KUKA KRL program: MyProgram_252().src

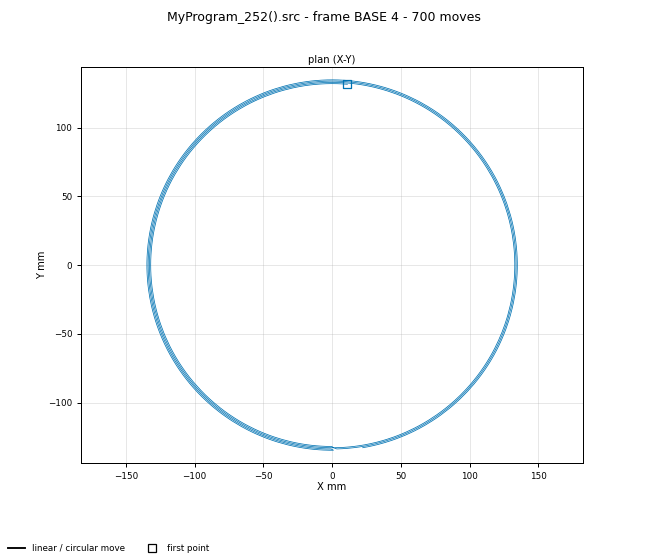
[picture p0: tool path of MyProgram_252().src in frame BASE 4, 700 of 700 moves have a stored position in this frame; points joined in program order, loops and branches not executed]
&ACCESS RVP
&REL 1
&PARAM TEMPLATE = C:\KRC\Roboter\Template\vorgabe
&PARAM EDITMASK = *
DEF MyProgram_252()
; ---- Setting reference (Base) ----
$BASE = BASE_DATA[4]

; --------------------------
; ---- Setting tool (TCP) ----
$TOOL = TOOL_DATA[3]
; --------------------------

$VEL.CP = VEL_APROX_PRINT
Startdeposition()
$VEL.CP = VEL_PRINT
LIN {X 11.0837,Y 131.5095,Z 165,A 85.1709,B 12.0272,C -0.0775,E1 12.0407,E2 365.1861} C_DIS
LIN {X 7.4461,Y 131.7673,Z 165,A 86.8868,B 12.0272,C -0.081,E1 12.0359,E2 363.4553} C_DIS
LIN {X 3.723,Y 131.9233,Z 165,A 88.4232,B 12.0272,C -0.079,E1 12.0316,E2 361.9291} C_DIS
LIN {X -0.4485,Y 131.9754,Z 165,A 90.2531,B 12.0272,C -0.0794,E1 12.0265,E2 360.0978} C_DIS
LIN {X -4.4864,Y 131.9012,Z 165,A 92.0505,B 12.0272,C -0.0802,E1 12.0215,E2 358.2962} C_DIS
LIN {X -8.3856,Y 131.7094,Z 165,A 93.7167,B 12.0272,C -0.0792,E1 12.0168,E2 356.6341} C_DIS
LIN {X -12.6017,Y 131.3727,Z 165,A 95.4316,B 12.0272,C -0.0756,E1 12.0121,E2 354.9346} C_DIS
LIN {X -16.1343,Y 130.9867,Z 165,A 97.1454,B 12.0272,C -0.0791,E1 12.0073,E2 353.2016} C_DIS
LIN {X -20.1878,Y 130.4225,Z 165,A 98.8102,B 12.0272,C -0.0756,E1 12.0027,E2 351.551} C_DIS
LIN {X -24.054,Y 129.7672,Z 165,A 100.47,B 12.0272,C -0.0736,E1 11.9982,E2 349.8973} C_DIS
LIN {X -28.8561,Y 128.7834,Z 165,A 102.7397,B 12.0272,C -0.0755,E1 11.992,E2 347.6125} C_DIS
LIN {X -32.281,Y 127.9668,Z 165,A 104.1599,B 12.0272,C -0.0718,E1 11.9881,E2 346.206} C_DIS
LIN {X -35.1769,Y 127.2017,Z 165,A 105.5524,B 12.0272,C -0.0729,E1 11.9844,E2 344.8037} C_DIS
LIN {X -39.2512,Y 126.0051,Z 165,A 107.686,B 12.0272,C -0.078,E1 11.9786,E2 342.6373} C_DIS
LIN {X -42.5812,Y 124.9193,Z 165,A 109.0037,B 12.0272,C -0.0717,E1 11.9752,E2 341.3448} C_DIS
LIN {X -46.1148,Y 123.6566,Z 165,A 110.4652,B 12.0272,C -0.066,E1 11.9714,E2 339.9042} C_DIS
LIN {X -48.8551,Y 122.6008,Z 165,A 111.8686,B 12.0272,C -0.0676,E1 11.9677,E2 338.4868} C_DIS
LIN {X -52.264,Y 121.1857,Z 165,A 113.1827,B 12.0273,C -0.0589,E1 11.9644,E2 337.2079} C_DIS
LIN {X -56.5408,Y 119.2509,Z 165,A 115.4801,B 12.0273,C -0.0623,E1 11.9585,E2 334.8819} C_DIS
LIN {X -59.5908,Y 117.7562,Z 165,A 116.8588,B 12.0273,C -0.0581,E1 11.9551,E2 333.5157} C_DIS
LIN {X -62.7217,Y 116.121,Z 165,A 118.4505,B 12.0273,C -0.0572,E1 11.9511,E2 331.9187} C_DIS
LIN {X -67.9902,Y 113.117,Z 165,A 121.2132,B 12.0273,C -0.0561,E1 11.9444,E2 329.1433} C_DIS
LIN {X -71.6438,Y 110.8388,Z 165,A 123.1109,B 12.0273,C -0.0537,E1 11.94,E2 327.2441} C_DIS
LIN {X -75.266,Y 108.4115,Z 165,A 124.9825,B 12.0273,C -0.05,E1 11.9357,E2 325.3769} C_DIS
LIN {X -78.4972,Y 106.096,Z 165,A 126.7552,B 12.0273,C -0.0479,E1 11.9316,E2 323.6005} C_DIS
LIN {X -81.8052,Y 103.5666,Z 165,A 128.5795,B 12.0273,C -0.0449,E1 11.9276,E2 321.7761} C_DIS
LIN {X -85.127,Y 100.8541,Z 165,A 130.4754,B 12.0274,C -0.0421,E1 11.9236,E2 319.878} C_DIS
LIN {X -88.4867,Y 97.9193,Z 165,A 132.4238,B 12.0274,C -0.0384,E1 11.9195,E2 317.9304} C_DIS
LIN {X -91.8671,Y 94.7546,Z 165,A 134.4232,B 12.0274,C -0.034,E1 11.9155,E2 315.9344} C_DIS
LIN {X -95.0357,Y 91.5768,Z 165,A 136.3955,B 12.0274,C -0.0303,E1 11.9116,E2 313.9614} C_DIS
LIN {X -98.0268,Y 88.3681,Z 165,A 138.3281,B 12.0274,C -0.0267,E1 11.908,E2 312.0276} C_DIS
LIN {X -100.8093,Y 85.18,Z 165,A 140.1811,B 12.0274,C -0.0229,E1 11.9046,E2 310.1748} C_DIS
LIN {X -103.4592,Y 81.9408,Z 165,A 142.0058,B 12.0274,C -0.0188,E1 11.9014,E2 308.3512} C_DIS
LIN {X -105.9833,Y 78.6485,Z 165,A 143.8053,B 12.0274,C -0.0144,E1 11.8984,E2 306.554} C_DIS
LIN {X -108.372,Y 75.3227,Z 165,A 145.6652,B 12.0274,C -0.0118,E1 11.8954,E2 304.6864} C_DIS
LIN {X -110.1166,Y 72.7488,Z 165,A 146.9884,B 12.0274,C -0.0079,E1 11.8933,E2 303.3679} C_DIS
LIN {X -114.2601,Y 66.0503,Z 165,A 150.4645,B 12.0274,C -0.0003,E1 11.8883,E2 299.8893} C_DIS
LIN {X -116.453,Y 62.1037,Z 165,A 152.4054,B 12.0274,C 0.0053,E1 11.8857,E2 297.953} C_DIS
LIN {X -118.178,Y 58.7502,Z 165,A 154.1788,B 12.0274,C 0.0066,E1 11.8835,E2 296.1653} C_DIS
LIN {X -120.2539,Y 54.3762,Z 165,A 155.9913,B 12.0274,C 0.0187,E1 11.8814,E2 294.3894} C_DIS
LIN {X -122.0747,Y 50.158,Z 165,A 158.225,B 12.0274,C 0.019,E1 11.8789,E2 292.1299} C_DIS
LIN {X -123.4373,Y 46.7004,Z 165,A 159.761,B 12.0274,C 0.0251,E1 11.8774,E2 290.605} C_DIS
LIN {X -124.6007,Y 43.5,Z 165,A 161.3273,B 12.0274,C 0.0274,E1 11.8759,E2 289.03} C_DIS
LIN {X -125.7157,Y 40.163,Z 165,A 162.8507,B 12.0274,C 0.0318,E1 11.8746,E2 287.5089} C_DIS
LIN {X -126.8783,Y 36.3323,Z 165,A 164.7046,B 12.0274,C 0.0343,E1 11.8731,E2 285.6434} C_DIS
LIN {X -127.9048,Y 32.5256,Z 165,A 166.3572,B 12.0274,C 0.0405,E1 11.872,E2 283.9996} C_DIS
LIN {X -129.1975,Y 26.9439,Z 165,A 168.886,B 12.0274,C 0.0468,E1 11.8704,E2 281.4689} C_DIS
LIN {X -129.8924,Y 23.3569,Z 165,A 170.4298,B 12.0274,C 0.0523,E1 11.8696,E2 279.9319} C_DIS
LIN {X -130.5188,Y 19.5658,Z 165,A 172.6918,B 12.0274,C 0.0443,E1 11.8687,E2 277.6013} C_DIS
LIN {X -131.1264,Y 14.9637,Z 165,A 174.1798,B 12.0274,C 0.0617,E1 11.8682,E2 276.1783} C_DIS
LIN {X -131.4859,Y 11.3639,Z 165,A 175.7627,B 12.0273,C 0.0661,E1 11.8678,E2 274.5957} C_DIS
LIN {X -131.7479,Y 7.761,Z 165,A 177.3281,B 12.0273,C 0.0708,E1 11.8675,E2 273.0324} C_DIS
LIN {X -131.9173,Y 3.9418,Z 165,A 178.9769,B 12.0273,C 0.0759,E1 11.8673,E2 271.3867} C_DIS
LIN {X -131.9786,Y 0.1809,Z 165,A -179.158,B 12.0273,C 0.0758,E1 11.8673,E2 269.4959} C_DIS
LIN {X -131.9226,Y -3.75,Z 165,A -177.5567,B 12.0272,C 0.0831,E1 11.8673,E2 267.9089} C_DIS
LIN {X -131.7465,Y -7.7839,Z 165,A -175.747,B 12.0272,C 0.087,E1 11.8676,E2 266.0943} C_DIS
LIN {X -131.4331,Y -11.9728,Z 165,A -173.8969,B 12.0272,C 0.0918,E1 11.8681,E2 264.243} C_DIS
LIN {X -130.9432,Y -16.4897,Z 165,A -171.415,B 12.0272,C 0.0864,E1 11.8689,E2 261.7023} C_DIS
LIN {X -130.292,Y -21.0255,Z 165,A -169.881,B 12.027,C 0.1022,E1 11.8696,E2 260.2248} C_DIS
LIN {X -129.8228,Y -23.746,Z 165,A -168.2147,B 12.0271,C 0.0954,E1 11.8705,E2 258.5036} C_DIS
LIN {X -128.9625,Y -28.0404,Z 165,A -166.7904,B 12.027,C 0.1113,E1 11.8712,E2 257.1383} C_DIS
LIN {X -127.9745,Y -32.2507,Z 165,A -164.9477,B 12.027,C 0.1174,E1 11.8724,E2 255.3015} C_DIS
LIN {X -127.1733,Y -35.2784,Z 165,A -163.2883,B 12.027,C 0.1147,E1 11.8737,E2 253.6076} C_DIS
LIN {X -125.8916,Y -39.6125,Z 165,A -161.4971,B 12.0268,C 0.1239,E1 11.8751,E2 251.8386} C_DIS
LIN {X -124.8136,Y -42.8859,Z 165,A -160.1385,B 12.0268,C 0.1311,E1 11.8763,E2 250.4977} C_DIS
LIN {X -123.7267,Y -45.9277,Z 165,A -158.7269,B 12.0268,C 0.1347,E1 11.8777,E2 249.0862} C_DIS
LIN {X -122.5757,Y -48.9172,Z 165,A -157.1757,B 12.0268,C 0.1349,E1 11.8793,E2 247.517} C_DIS
LIN {X -121.1996,Y -52.2318,Z 165,A -155.4885,B 12.0268,C 0.1362,E1 11.8811,E2 245.8156} C_DIS
LIN {X -118.0518,Y -59.0061,Z 165,A -152.363,B 12.0266,C 0.1474,E1 11.8849,E2 242.7068} C_DIS
LIN {X -116.1071,Y -62.7476,Z 165,A -150.4309,B 12.0266,C 0.1498,E1 11.8874,E2 240.764} C_DIS
LIN {X -113.9846,Y -66.5256,Z 165,A -148.5372,B 12.0266,C 0.1542,E1 11.89,E2 238.8701} C_DIS
LIN {X -111.9038,Y -69.9687,Z 165,A -146.721,B 12.0265,C 0.157,E1 11.8927,E2 237.0467} C_DIS
LIN {X -109.4503,Y -73.7476,Z 165,A -144.6081,B 12.0265,C 0.1581,E1 11.896,E2 234.9162} C_DIS
LIN {X -106.573,Y -77.8481,Z 165,A -142.5388,B 12.0264,C 0.1656,E1 11.8993,E2 232.8609} C_DIS
LIN {X -103.9034,Y -81.3764,Z 165,A -140.7404,B 12.0263,C 0.1727,E1 11.9024,E2 231.0783} C_DIS
LIN {X -101.0773,Y -84.861,Z 165,A -138.7731,B 12.0262,C 0.1766,E1 11.9059,E2 229.1097} C_DIS
LIN {X -95.5361,Y -91.0543,Z 165,A -135.0199,B 12.0262,C 0.1809,E1 11.913,E2 225.3409} C_DIS
LIN {X -92.3052,Y -94.328,Z 165,A -133.0328,B 12.0261,C 0.1851,E1 11.9169,E2 223.3559} C_DIS
LIN {X -89.3699,Y -97.1134,Z 165,A -131.2465,B 12.0261,C 0.1878,E1 11.9205,E2 221.5667} C_DIS
LIN {X -86.0304,Y -100.0839,Z 165,A -128.5328,B 12.0262,C 0.1733,E1 11.9265,E2 218.7596} C_DIS
LIN {X -81.3334,Y -103.9372,Z 165,A -126.6263,B 12.0259,C 0.195,E1 11.9305,E2 216.943} C_DIS
LIN {X -78.4155,Y -106.1561,Z 165,A -125.0015,B 12.0259,C 0.1969,E1 11.9341,E2 215.3146} C_DIS
LIN {X -75.3351,Y -108.3634,Z 165,A -123.2252,B 12.0259,C 0.1964,E1 11.9382,E2 213.5228} C_DIS
LIN {X -70.9431,Y -111.2886,Z 165,A -121.1913,B 12.0257,C 0.206,E1 11.9429,E2 211.5205} C_DIS
LIN {X -67.7985,Y -113.2318,Z 165,A -119.5058,B 12.0257,C 0.2063,E1 11.9469,E2 209.8255} C_DIS
LIN {X -64.4281,Y -115.1829,Z 165,A -117.8448,B 12.0257,C 0.2093,E1 11.9509,E2 208.1683} C_DIS
LIN {X -61.2678,Y -116.892,Z 165,A -116.2912,B 12.0257,C 0.2114,E1 11.9548,E2 206.6155} C_DIS
LIN {X -56.087,Y -119.4668,Z 165,A -113.7169,B 12.0257,C 0.2129,E1 11.9612,E2 204.0338} C_DIS
LIN {X -52.5475,Y -121.0631,Z 165,A -112.0714,B 12.0256,C 0.2157,E1 11.9654,E2 202.3931} C_DIS
LIN {X -49.413,Y -122.3759,Z 165,A -110.5286,B 12.0256,C 0.2155,E1 11.9694,E2 200.8422} C_DIS
LIN {X -45.5639,Y -123.863,Z 165,A -108.7403,B 12.0256,C 0.2173,E1 11.9741,E2 199.0541} C_DIS
LIN {X -41.8431,Y -125.1667,Z 165,A -107.0564,B 12.0256,C 0.2194,E1 11.9785,E2 197.3734} C_DIS
LIN {X -36.3101,Y -126.8847,Z 165,A -104.4227,B 12.0256,C 0.2183,E1 11.9856,E2 194.7251} C_DIS
LIN {X -30.1061,Y -128.4979,Z 165,A -101.6536,B 12.0255,C 0.2203,E1 11.9931,E2 191.9571} C_DIS
LIN {X -26.2294,Y -129.3429,Z 165,A -100.0343,B 12.0255,C 0.2237,E1 11.9975,E2 190.3499} C_DIS
LIN {X -22.4415,Y -130.0557,Z 165,A -98.2616,B 12.0255,C 0.2219,E1 12.0024,E2 188.5647} C_DIS
LIN {X -19.0063,Y -130.6004,Z 165,A -96.7818,B 12.0255,C 0.2231,E1 12.0065,E2 187.088} C_DIS
LIN {X -15.4939,Y -131.0631,Z 165,A -95.2317,B 12.0255,C 0.2231,E1 12.0108,E2 185.5359} C_DIS
LIN {X -11.5691,Y -131.4685,Z 165,A -93.6029,B 12.0254,C 0.2255,E1 12.0153,E2 183.9167} C_DIS
LIN {X -8.1546,Y -131.7236,Z 165,A -92.0385,B 12.0254,C 0.2236,E1 12.0197,E2 182.3422} C_DIS
LIN {X -4.1808,Y -131.9106,Z 165,A -90.2808,B 12.0254,C 0.2228,E1 12.0246,E2 180.5801} C_DIS
LIN {X -0.1658,Y -131.977,Z 165,A -88.5589,B 12.0254,C 0.2231,E1 12.0294,E2 178.86} C_DIS
LIN {X -0.1658,Y -131.977,Z 165,A -88.5589,B 12.0254,C 0.2231,E1 12.0294,E2 178.86} C_DIS
Enddeposition()
LIN {X 0.9669,Y -132.8884,Z 165,A -88.2437,B 12.0251,C 0.2348,E1 12.03,E2 178.6008} C_DIS
Startdeposition()
$VEL.CP = VEL_PRINT
LIN {X -1.6364,Y -132.8852,Z 165,A -89.9774,B 12.0248,C 0.2505,E1 12.025,E2 180.4097} C_DIS
LIN {X -5.3601,Y -132.7859,Z 165,A -91.5116,B 12.0248,C 0.2487,E1 12.0207,E2 181.9358} C_DIS
LIN {X -9.7113,Y -132.5386,Z 165,A -93.3724,B 12.0248,C 0.2482,E1 12.0156,E2 183.7952} C_DIS
LIN {X -13.4707,Y -132.2115,Z 165,A -95.1283,B 12.0248,C 0.2512,E1 12.0106,E2 185.5674} C_DIS
LIN {X -17.4667,Y -131.7411,Z 165,A -96.7577,B 12.0248,C 0.2482,E1 12.0061,E2 187.1846} C_DIS
LIN {X -21.5719,Y -131.1316,Z 165,A -98.5371,B 12.0248,C 0.2473,E1 12.0012,E2 188.9633} C_DIS
LIN {X -25.059,Y -130.5098,Z 165,A -100.049,B 12.0248,C 0.2464,E1 11.9971,E2 190.4738} C_DIS
LIN {X -28.736,Y -129.7516,Z 165,A -101.8197,B 12.0248,C 0.2493,E1 11.9922,E2 192.2633} C_DIS
LIN {X -33.8948,Y -128.499,Z 165,A -104.0819,B 12.0248,C 0.2473,E1 11.9861,E2 194.5228} C_DIS
LIN {X -37.8678,Y -127.3854,Z 165,A -105.8921,B 12.0248,C 0.2468,E1 11.9812,E2 196.337} C_DIS
LIN {X -41.8336,Y -126.1375,Z 165,A -107.5265,B 12.025,C 0.2416,E1 11.9769,E2 197.9525} C_DIS
LIN {X -45.0896,Y -125.0105,Z 165,A -109.037,B 12.025,C 0.2409,E1 11.9729,E2 199.4662} C_DIS
LIN {X -48.2888,Y -123.8099,Z 165,A -110.496,B 12.025,C 0.2392,E1 11.9691,E2 200.9235} C_DIS
LIN {X -51.3805,Y -122.5592,Z 165,A -111.9768,B 12.025,C 0.2388,E1 11.9653,E2 202.4095} C_DIS
LIN {X -54.4734,Y -121.2162,Z 165,A -113.4617,B 12.025,C 0.238,E1 11.9615,E2 203.8982} C_DIS
LIN {X -58.4379,Y -119.3559,Z 165,A -115.4331,B 12.025,C 0.2378,E1 11.9565,E2 205.8796} C_DIS
LIN {X -61.8393,Y -117.6289,Z 165,A -116.9935,B 12.0251,C 0.2337,E1 11.9527,E2 207.4296} C_DIS
LIN {X -65.5899,Y -115.5822,Z 165,A -118.9368,B 12.0251,C 0.2337,E1 11.9479,E2 209.385} C_DIS
LIN {X -70.5677,Y -112.6125,Z 165,A -121.3868,B 12.0252,C 0.229,E1 11.9421,E2 211.8288} C_DIS
LIN {X -74.0604,Y -110.3465,Z 165,A -123.3411,B 12.0252,C 0.23,E1 11.9374,E2 213.8019} C_DIS
LIN {X -77.5478,Y -107.9241,Z 165,A -125.115,B 12.0252,C 0.2258,E1 11.9334,E2 215.5685} C_DIS
LIN {X -80.4326,Y -105.7919,Z 165,A -126.629,B 12.0254,C 0.2224,E1 11.9301,E2 217.0782} C_DIS
LIN {X -83.8323,Y -103.1186,Z 165,A -128.8268,B 12.0253,C 0.2268,E1 11.9252,E2 219.3153} C_DIS
LIN {X -86.6745,Y -100.7408,Z 165,A -129.86,B 12.0256,C 0.2109,E1 11.9231,E2 220.2803} C_DIS
LIN {X -88.9595,Y -98.7297,Z 165,A -131.4614,B 12.0255,C 0.2151,E1 11.9197,E2 221.916} C_DIS
LIN {X -92.0207,Y -95.8825,Z 165,A -133.2607,B 12.0255,C 0.2116,E1 11.9161,E2 223.7142} C_DIS
LIN {X -95.158,Y -92.7701,Z 165,A -135.1993,B 12.0256,C 0.2085,E1 11.9122,E2 225.656} C_DIS
LIN {X -98.3035,Y -89.4294,Z 165,A -137.5582,B 12.0256,C 0.213,E1 11.9077,E2 228.0593} C_DIS
LIN {X -101.0067,Y -86.3653,Z 165,A -138.8103,B 12.0258,C 0.1977,E1 11.9055,E2 229.2498} C_DIS
LIN {X -103.1749,Y -83.7633,Z 165,A -140.4648,B 12.0258,C 0.1989,E1 11.9026,E2 230.9266} C_DIS
LIN {X -105.9003,Y -80.2895,Z 165,A -142.4027,B 12.0258,C 0.1953,E1 11.8992,E2 232.8676} C_DIS
LIN {X -108.5302,Y -76.6968,Z 165,A -144.5723,B 12.0258,C 0.1964,E1 11.8957,E2 235.0657} C_DIS
LIN {X -110.5325,Y -73.7818,Z 165,A -145.6225,B 12.026,C 0.1822,E1 11.8941,E2 236.0584} C_DIS
LIN {X -112.6635,Y -70.4857,Z 165,A -147.515,B 12.026,C 0.1826,E1 11.8912,E2 237.9739} C_DIS
LIN {X -114.7935,Y -66.9612,Z 165,A -149.3632,B 12.026,C 0.1798,E1 11.8886,E2 239.8295} C_DIS
LIN {X -116.8802,Y -63.2484,Z 165,A -151.2328,B 12.0261,C 0.1759,E1 11.8861,E2 241.7018} C_DIS
LIN {X -118.682,Y -59.7958,Z 165,A -152.8981,B 12.0261,C 0.1712,E1 11.884,E2 243.364} C_DIS
LIN {X -120.5344,Y -55.9658,Z 165,A -154.4185,B 12.0263,C 0.1595,E1 11.8822,E2 244.8456} C_DIS
LIN {X -121.5966,Y -53.6229,Z 165,A -155.7743,B 12.0263,C 0.162,E1 11.8806,E2 246.23} C_DIS
LIN {X -123.1001,Y -50.0721,Z 165,A -157.5682,B 12.0263,C 0.1604,E1 11.8786,E2 248.0382} C_DIS
LIN {X -124.4801,Y -46.5338,Z 165,A -159.1245,B 12.0264,C 0.1542,E1 11.8771,E2 249.5834} C_DIS
LIN {X -125.6277,Y -43.3406,Z 165,A -160.6042,B 12.0264,C 0.1505,E1 11.8757,E2 251.0639} C_DIS
LIN {X -126.7133,Y -40.0574,Z 165,A -162.2539,B 12.0264,C 0.1499,E1 11.8743,E2 252.7311} C_DIS
LIN {X -128.8623,Y -32.4851,Z 165,A -165.5463,B 12.0266,C 0.1381,E1 11.8719,E2 256.0083} C_DIS
LIN {X -129.7399,Y -28.7902,Z 165,A -167.6588,B 12.0266,C 0.1437,E1 11.8705,E2 258.1756} C_DIS
LIN {X -130.5159,Y -25.0267,Z 165,A -168.9735,B 12.0266,C 0.1315,E1 11.8699,E2 259.4482} C_DIS
LIN {X -131.4162,Y -19.7702,Z 165,A -171.4049,B 12.0267,C 0.1277,E1 11.8688,E2 261.893} C_DIS
LIN {X -132.0073,Y -15.3299,Z 165,A -173.2583,B 12.0267,C 0.1204,E1 11.8681,E2 263.7353} C_DIS
LIN {X -132.4193,Y -11.2216,Z 165,A -174.9858,B 12.0268,C 0.1141,E1 11.8677,E2 265.4546} C_DIS
LIN {X -132.6842,Y -7.4947,Z 165,A -176.7198,B 12.0268,C 0.112,E1 11.8674,E2 267.2015} C_DIS
LIN {X -132.8527,Y -3.3319,Z 165,A -178.5408,B 12.0269,C 0.1072,E1 11.8672,E2 269.0235} C_DIS
LIN {X -132.8939,Y 0.6025,Z 165,A 179.7573,B 12.0269,C 0.1023,E1 11.8672,E2 270.7243} C_DIS
LIN {X -132.7993,Y 5.017,Z 165,A 177.9002,B 12.027,C 0.0957,E1 11.8673,E2 272.5738} C_DIS
LIN {X -132.62,Y 8.5354,Z 165,A 176.3122,B 12.027,C 0.0927,E1 11.8676,E2 274.1682} C_DIS
LIN {X -132.3011,Y 12.5391,Z 165,A 174.6151,B 12.027,C 0.0868,E1 11.868,E2 275.8593} C_DIS
LIN {X -131.8994,Y 16.2346,Z 165,A 172.968,B 12.027,C 0.0831,E1 11.8685,E2 277.5099} C_DIS
LIN {X -130.8416,Y 23.2646,Z 165,A 169.7393,B 12.0271,C 0.0776,E1 11.87,E2 280.7543} C_DIS
LIN {X -129.8984,Y 28.0558,Z 165,A 167.27,B 12.0271,C 0.0793,E1 11.8714,E2 283.2638} C_DIS
LIN {X -128.9181,Y 32.2652,Z 165,A 166.0479,B 12.0272,C 0.0601,E1 11.8722,E2 284.4086} C_DIS
LIN {X -127.9808,Y 35.7998,Z 165,A 164.2862,B 12.0272,C 0.0596,E1 11.8734,E2 286.1902} C_DIS
LIN {X -127.0462,Y 38.9869,Z 165,A 162.8075,B 12.0272,C 0.0565,E1 11.8746,E2 287.6727} C_DIS
LIN {X -125.7951,Y 42.8579,Z 165,A 160.9368,B 12.0272,C 0.0541,E1 11.8763,E2 289.5552} C_DIS
LIN {X -124.4445,Y 46.629,Z 165,A 159.3402,B 12.0272,C 0.0464,E1 11.8778,E2 291.1344} C_DIS
LIN {X -123.1358,Y 49.9835,Z 165,A 157.7546,B 12.0273,C 0.0428,E1 11.8794,E2 292.7221} C_DIS
LIN {X -121.2066,Y 54.4949,Z 165,A 155.5761,B 12.0273,C 0.0384,E1 11.8819,E2 294.9055} C_DIS
LIN {X -118.7734,Y 59.6163,Z 165,A 153.1688,B 12.0273,C 0.031,E1 11.8848,E2 297.3056} C_DIS
LIN {X -116.5566,Y 63.8421,Z 165,A 150.5656,B 12.0273,C 0.0374,E1 11.8883,E2 299.9701} C_DIS
LIN {X -114.4892,Y 67.4793,Z 165,A 149.2931,B 12.0273,C 0.0212,E1 11.89,E2 301.1785} C_DIS
LIN {X -111.0541,Y 72.9943,Z 165,A 146.6881,B 12.0273,C 0.0098,E1 11.8939,E2 303.7573} C_DIS
LIN {X -108.206,Y 77.1537,Z 165,A 144.0936,B 12.0273,C 0.0137,E1 11.898,E2 306.3987} C_DIS
LIN {X -105.5046,Y 80.8083,Z 165,A 142.1364,B 12.0273,C 0.0089,E1 11.9013,E2 308.3535} C_DIS
LIN {X -102.8384,Y 84.1752,Z 165,A 140.2696,B 12.0273,C 0.0049,E1 11.9046,E2 310.22} C_DIS
LIN {X -99.9382,Y 87.5992,Z 165,A 138.3126,B 12.0273,C 0.001,E1 11.9081,E2 312.1774} C_DIS
LIN {X -96.9717,Y 90.8727,Z 165,A 136.3446,B 12.0273,C -0.0019,E1 11.9119,E2 314.1507} C_DIS
LIN {X -93.8909,Y 94.052,Z 165,A 134.4214,B 12.0273,C -0.0057,E1 11.9156,E2 316.0735} C_DIS
LIN {X -90.6399,Y 97.1885,Z 165,A 132.4789,B 12.0273,C -0.0098,E1 11.9196,E2 318.0133} C_DIS
LIN {X -87.2549,Y 100.2387,Z 165,A 130.5251,B 12.0273,C -0.014,E1 11.9236,E2 319.9637} C_DIS
LIN {X -83.8131,Y 103.1343,Z 165,A 128.5433,B 12.0273,C -0.0168,E1 11.9279,E2 321.9485} C_DIS
LIN {X -80.3503,Y 105.8544,Z 165,A 126.609,B 12.0273,C -0.0195,E1 11.9322,E2 323.885} C_DIS
LIN {X -76.857,Y 108.4172,Z 165,A 124.7384,B 12.0273,C -0.0228,E1 11.9364,E2 325.7541} C_DIS
LIN {X -73.2685,Y 110.8737,Z 165,A 122.8408,B 12.0273,C -0.0255,E1 11.9408,E2 327.6524} C_DIS
LIN {X -69.6079,Y 113.2076,Z 165,A 120.9734,B 12.0273,C -0.0286,E1 11.9452,E2 329.5175} C_DIS
LIN {X -65.7193,Y 115.5084,Z 165,A 118.2114,B 12.0273,C -0.0131,E1 11.9522,E2 332.3719} C_DIS
LIN {X -60.2277,Y 118.4622,Z 165,A 116.2852,B 12.0273,C -0.0343,E1 11.9567,E2 334.2074} C_DIS
LIN {X -52.6794,Y 122.0064,Z 165,A 112.8297,B 12.0273,C -0.0422,E1 11.9654,E2 337.6435} C_DIS
LIN {X -49.7383,Y 123.2346,Z 165,A 111.3701,B 12.0273,C -0.0418,E1 11.9692,E2 339.1121} C_DIS
LIN {X -46.1696,Y 124.6165,Z 165,A 109.7453,B 12.0273,C -0.0442,E1 11.9734,E2 340.7326} C_DIS
LIN {X -42.2829,Y 125.9879,Z 165,A 107.0728,B 12.0273,C -0.0252,E1 11.9808,E2 343.5074} C_DIS
LIN {X -36.2422,Y 127.8571,Z 165,A 105.3766,B 12.0273,C -0.0517,E1 11.985,E2 345.0822} C_DIS
LIN {X -32.1984,Y 128.935,Z 165,A 102.3456,B 12.0273,C -0.0243,E1 11.9936,E2 348.2541} C_DIS
LIN {X -25.1621,Y 130.4901,Z 165,A 100.5485,B 12.0273,C -0.0572,E1 11.9981,E2 349.8973} C_DIS
LIN {X -21.5719,Y 131.1316,Z 165,A 98.7353,B 12.0273,C -0.0524,E1 12.0032,E2 351.7378} C_DIS
LIN {X -18.2752,Y 131.6323,Z 165,A 97.1666,B 12.0273,C -0.0499,E1 12.0075,E2 353.3209} C_DIS
LIN {X -14.2264,Y 132.1302,Z 165,A 95.5011,B 12.0273,C -0.0529,E1 12.0121,E2 354.9744} C_DIS
LIN {X -10.2517,Y 132.4992,Z 165,A 93.7279,B 12.0273,C -0.0521,E1 12.0171,E2 356.7528} C_DIS
LIN {X -6.471,Y 132.7365,Z 165,A 92.1663,B 12.0273,C -0.0542,E1 12.0214,E2 358.3052} C_DIS
LIN {X -2.4477,Y 132.8717,Z 165,A 90.3952,B 12.0273,C -0.0536,E1 12.0264,E2 360.0796} C_DIS
LIN {X 1.5303,Y 132.8869,Z 165,A 88.6001,B 12.0273,C -0.0517,E1 12.0314,E2 361.8833} C_DIS
LIN {X 5.3663,Y 132.7857,Z 165,A 87.0553,B 12.0273,C -0.0544,E1 12.0357,E2 363.4145} C_DIS
LIN {X 9.3782,Y 132.5629,Z 165,A 85.2795,B 12.0273,C -0.0531,E1 12.0406,E2 365.1947} C_DIS
LIN {X 13.0895,Y 132.2482,Z 165,A 83.638,B 12.0273,C -0.0519,E1 12.0452,E2 366.8398} C_DIS
LIN {X 17.1232,Y 131.7861,Z 165,A 81.9542,B 12.0273,C -0.053,E1 12.0498,E2 368.5151} C_DIS
LIN {X 20.5913,Y 131.2891,Z 165,A 80.4758,B 12.0273,C -0.0532,E1 12.0539,E2 369.9893} C_DIS
LIN {X 24.4169,Y 130.6325,Z 165,A 78.7087,B 12.0273,C -0.0501,E1 12.0588,E2 371.767} C_DIS
LIN {X 28.2175,Y 129.8635,Z 165,A 76.8358,B 12.0273,C -0.0442,E1 12.064,E2 373.663} C_DIS
LIN {X 31.354,Y 129.1422,Z 165,A 75.6142,B 12.0273,C -0.0474,E1 12.0672,E2 374.8649} C_DIS
LIN {X 36.432,Y 127.804,Z 165,A 73.2336,B 12.0273,C -0.0429,E1 12.0737,E2 377.2588} C_DIS
LIN {X 40.5585,Y 126.5533,Z 165,A 71.654,B 12.0273,C -0.0484,E1 12.0778,E2 378.8054} C_DIS
LIN {X 43.6968,Y 125.5042,Z 165,A 70.2156,B 12.0273,C -0.0469,E1 12.0816,E2 380.245} C_DIS
LIN {X 46.7214,Y 124.4098,Z 165,A 68.8706,B 12.0273,C -0.0466,E1 12.0851,E2 381.585} C_DIS
LIN {X 49.9959,Y 123.1308,Z 165,A 67.3318,B 12.0273,C -0.0444,E1 12.0891,E2 383.1265} C_DIS
LIN {X 53.0238,Y 121.8575,Z 165,A 65.8769,B 12.0273,C -0.0419,E1 12.0929,E2 384.586} C_DIS
LIN {X 57.0972,Y 120.0025,Z 165,A 63.9663,B 12.0273,C -0.0401,E1 12.0977,E2 386.4943} C_DIS
LIN {X 60.7982,Y 118.1717,Z 165,A 62.2135,B 12.0273,C -0.0385,E1 12.1021,E2 388.2441} C_DIS
LIN {X 64.5473,Y 116.1674,Z 165,A 60.0014,B 12.0273,C -0.0262,E1 12.1076,E2 390.501} C_DIS
LIN {X 67.8292,Y 114.2823,Z 165,A 58.8108,B 12.0273,C -0.0353,E1 12.1104,E2 391.6399} C_DIS
LIN {X 71.1876,Y 112.2212,Z 165,A 56.9799,B 12.0273,C -0.0293,E1 12.1147,E2 393.4868} C_DIS
LIN {X 74.9013,Y 109.7776,Z 165,A 55.0661,B 12.0273,C -0.0263,E1 12.1192,E2 395.4006} C_DIS
LIN {X 78.4543,Y 107.2669,Z 165,A 53.2081,B 12.0273,C -0.0237,E1 12.1234,E2 397.257} C_DIS
LIN {X 82.0603,Y 104.5337,Z 165,A 51.2978,B 12.0273,C -0.0213,E1 12.1276,E2 399.1631} C_DIS
LIN {X 85.638,Y 101.6238,Z 165,A 49.3391,B 12.0273,C -0.0185,E1 12.1318,E2 401.1189} C_DIS
LIN {X 88.9555,Y 98.7332,Z 165,A 47.4128,B 12.0273,C -0.0141,E1 12.1358,E2 403.0494} C_DIS
LIN {X 92.1718,Y 95.7376,Z 165,A 45.5275,B 12.0273,C -0.0106,E1 12.1397,E2 404.9343} C_DIS
LIN {X 95.3263,Y 92.5965,Z 165,A 43.6368,B 12.0273,C -0.0074,E1 12.1434,E2 406.8225} C_DIS
LIN {X 98.4976,Y 89.2156,Z 165,A 41.6991,B 12.0273,C -0.0048,E1 12.147,E2 408.7538} C_DIS
LIN {X 101.4594,Y 85.8328,Z 165,A 39.7688,B 12.0273,C -0.0008,E1 12.1505,E2 410.6842} C_DIS
LIN {X 104.1879,Y 82.4995,Z 165,A 37.935,B 12.0273,C 0.0028,E1 12.1538,E2 412.5162} C_DIS
LIN {X 106.8542,Y 79.016,Z 165,A 36.0979,B 12.0273,C 0.0057,E1 12.1568,E2 414.348} C_DIS
LIN {X 109.8755,Y 74.7574,Z 165,A 34.1117,B 12.0273,C 0.0038,E1 12.16,E2 416.304} C_DIS
LIN {X 112.5366,Y 70.6879,Z 165,A 31.7528,B 12.0273,C 0.0161,E1 12.1636,E2 418.6956} C_DIS
LIN {X 116.3459,Y 64.2251,Z 165,A 28.7826,B 12.0273,C 0.017,E1 12.1677,E2 421.6366} C_DIS
LIN {X 117.7394,Y 61.6288,Z 165,A 26.8399,B 12.0273,C 0.0387,E1 12.1704,E2 423.6601} C_DIS
LIN {X 119.7761,Y 57.5713,Z 165,A 25.6457,B 12.0273,C 0.0229,E1 12.1717,E2 424.7651} C_DIS
LIN {X 121.5591,Y 53.7067,Z 165,A 23.621,B 12.0273,C 0.033,E1 12.1741,E2 426.8139} C_DIS
LIN {X 123.097,Y 50.0799,Z 165,A 21.7705,B 12.0273,C 0.0418,E1 12.1761,E2 428.6839} C_DIS
LIN {X 124.9887,Y 45.15,Z 165,A 19.6745,B 12.0273,C 0.043,E1 12.1781,E2 430.7603} C_DIS
LIN {X 126.1244,Y 41.8731,Z 165,A 17.6819,B 12.0273,C 0.0609,E1 12.18,E2 432.8134} C_DIS
LIN {X 127.481,Y 37.5413,Z 165,A 15.5908,B 12.0272,C 0.0702,E1 12.1816,E2 434.9222} C_DIS
LIN {X 128.8947,Y 32.3575,Z 165,A 14.0479,B 12.0272,C 0.0553,E1 12.1826,E2 436.3751} C_DIS
LIN {X 129.6644,Y 29.1222,Z 165,A 12.6402,B 12.0272,C 0.0586,E1 12.1835,E2 437.7811} C_DIS
LIN {X 130.2643,Y 26.3056,Z 165,A 11.3186,B 12.0272,C 0.0644,E1 12.1843,E2 439.1135} C_DIS
LIN {X 131.0478,Y 22.0743,Z 165,A 9.5249,B 12.0272,C 0.0681,E1 12.1851,E2 440.9016} C_DIS
LIN {X 131.5815,Y 18.631,Z 165,A 8.08,B 12.0272,C 0.0709,E1 12.1857,E2 442.3411} C_DIS
LIN {X 131.9753,Y 15.5986,Z 165,A 6.7469,B 12.0272,C 0.0751,E1 12.1862,E2 443.6773} C_DIS
LIN {X 132.3833,Y 11.6479,Z 165,A 4.9898,B 12.0272,C 0.0814,E1 12.1867,E2 445.4416} C_DIS
LIN {X 132.6429,Y 8.1647,Z 165,A 3.5534,B 12.0271,C 0.0839,E1 12.1869,E2 446.8712} C_DIS
LIN {X 132.804,Y 4.8961,Z 165,A 2.178,B 12.0271,C 0.0871,E1 12.1871,E2 448.2438} C_DIS
LIN {X 132.8903,Y 1.1306,Z 165,A 0.5737,B 12.0271,C 0.0913,E1 12.1871,E2 449.8476} C_DIS
LIN {X 132.8672,Y -2.7135,Z 165,A -1.1396,B 12.027,C 0.0978,E1 12.1871,E2 451.5694} C_DIS
LIN {X 132.7289,Y -6.6207,Z 165,A -2.7313,B 12.027,C 0.1001,E1 12.1869,E2 453.1516} C_DIS
LIN {X 132.4953,Y -10.305,Z 165,A -4.4267,B 12.027,C 0.1078,E1 12.1866,E2 454.8613} C_DIS
LIN {X 132.1415,Y -14.121,Z 165,A -5.945,B 12.0269,C 0.1089,E1 12.1862,E2 456.3652} C_DIS
LIN {X 131.7263,Y -17.5794,Z 165,A -7.4408,B 12.0269,C 0.1131,E1 12.1857,E2 457.8621} C_DIS
LIN {X 131.109,Y -21.7076,Z 165,A -9.218,B 12.0269,C 0.1178,E1 12.1849,E2 459.6387} C_DIS
LIN {X 130.5114,Y -25.0504,Z 165,A -10.6742,B 12.0268,C 0.1219,E1 12.1842,E2 461.0955} C_DIS
LIN {X 129.6726,Y -29.0862,Z 165,A -12.5338,B 12.0267,C 0.1294,E1 12.183,E2 462.9672} C_DIS
LIN {X 127.8249,Y -36.3574,Z 165,A -15.5263,B 12.0267,C 0.1319,E1 12.181,E2 465.9343} C_DIS
LIN {X 127.0711,Y -38.9055,Z 165,A -17.3413,B 12.0264,C 0.1539,E1 12.1794,E2 467.8312} C_DIS
LIN {X 125.5501,Y -43.5645,Z 165,A -18.4841,B 12.0267,C 0.1327,E1 12.1785,E2 468.8594} C_DIS
LIN {X 123.6469,Y -48.7082,Z 165,A -21.1249,B 12.0265,C 0.1472,E1 12.1759,E2 471.5366} C_DIS
LIN {X 122.5034,Y -51.514,Z 165,A -22.4443,B 12.0265,C 0.1512,E1 12.1745,E2 472.8591} C_DIS
LIN {X 121.1647,Y -54.5886,Z 165,A -24.148,B 12.0263,C 0.1624,E1 12.1725,E2 474.5958} C_DIS
LIN {X 118.2016,Y -60.7395,Z 165,A -26.7453,B 12.0263,C 0.1607,E1 12.1693,E2 477.1546} C_DIS
LIN {X 116.7166,Y -63.5486,Z 165,A -28.3209,B 12.0262,C 0.1701,E1 12.1672,E2 478.7568} C_DIS
LIN {X 114.5191,Y -67.4284,Z 165,A -29.9563,B 12.0262,C 0.1671,E1 12.165,E2 480.3598} C_DIS
LIN {X 112.637,Y -70.5282,Z 165,A -31.6494,B 12.0262,C 0.1748,E1 12.1625,E2 482.0704} C_DIS
LIN {X 110.4141,Y -73.9591,Z 165,A -33.3857,B 12.0261,C 0.1785,E1 12.1598,E2 483.8056} C_DIS
LIN {X 108.0253,Y -77.4063,Z 165,A -35.1776,B 12.0261,C 0.1825,E1 12.1569,E2 485.5976} C_DIS
LIN {X 105.5493,Y -80.7497,Z 165,A -36.983,B 12.0259,C 0.1872,E1 12.1539,E2 487.4065} C_DIS
LIN {X 102.7009,Y -84.3434,Z 165,A -39.2897,B 12.0257,C 0.201,E1 12.1498,E2 489.7554} C_DIS
LIN {X 100.14,Y -87.368,Z 165,A -40.5908,B 12.0258,C 0.1938,E1 12.1475,E2 491.0091} C_DIS
LIN {X 97.3535,Y -90.4627,Z 165,A -42.4198,B 12.0258,C 0.1988,E1 12.144,E2 492.8442} C_DIS
LIN {X 93.2409,Y -94.6963,Z 165,A -45.0926,B 12.0256,C 0.2079,E1 12.1387,E2 495.5354} C_DIS
LIN {X 89.4924,Y -98.2464,Z 165,A -47.1594,B 12.0256,C 0.2082,E1 12.1345,E2 497.5853} C_DIS
LIN {X 86.2368,Y -101.116,Z 165,A -49.3072,B 12.0254,C 0.2195,E1 12.1299,E2 499.7685} C_DIS
LIN {X 83.3123,Y -103.5387,Z 165,A -50.7256,B 12.0254,C 0.2168,E1 12.1269,E2 501.1622} C_DIS
LIN {X 79.7827,Y -106.2827,Z 165,A -52.5102,B 12.0254,C 0.2166,E1 12.123,E2 502.9316} C_DIS
LIN {X 76.2834,Y -108.8218,Z 165,A -54.3684,B 12.0254,C 0.2198,E1 12.1187,E2 504.7909} C_DIS
LIN {X 70.5979,Y -112.5934,Z 165,A -57.332,B 12.0253,C 0.2255,E1 12.1118,E2 507.7601} C_DIS
LIN {X 66.8243,Y -114.8729,Z 165,A -59.164,B 12.0253,C 0.2267,E1 12.1074,E2 509.5856} C_DIS
LIN {X 63.1793,Y -116.9174,Z 165,A -60.9618,B 12.0253,C 0.2294,E1 12.103,E2 511.3847} C_DIS
LIN {X 60.1113,Y -118.5214,Z 165,A -62.374,B 12.0253,C 0.2294,E1 12.0995,E2 512.7883} C_DIS
LIN {X 56.7026,Y -120.1911,Z 165,A -63.9919,B 12.0252,C 0.2313,E1 12.0955,E2 514.4056} C_DIS
LIN {X 53.9423,Y -121.4538,Z 165,A -65.2668,B 12.0252,C 0.2321,E1 12.0922,E2 515.6775} C_DIS
LIN {X 50.9073,Y -122.7568,Z 165,A -66.6995,B 12.0252,C 0.2341,E1 12.0885,E2 517.1125} C_DIS
LIN {X 47.8283,Y -123.9889,Z 165,A -68.1466,B 12.0251,C 0.2363,E1 12.0848,E2 518.5628} C_DIS
LIN {X 44.4901,Y -125.2266,Z 165,A -70.3388,B 12.0247,C 0.2553,E1 12.0788,E2 520.8358} C_DIS
LIN {X 39.5333,Y -126.8789,Z 165,A -71.8407,B 12.0251,C 0.238,E1 12.075,E2 522.2488} C_DIS
LIN {X 36.3429,Y -127.8289,Z 165,A -73.8534,B 12.0247,C 0.2544,E1 12.0694,E2 524.3325} C_DIS
LIN {X 32.0909,Y -128.9623,Z 165,A -75.3708,B 12.0249,C 0.2462,E1 12.0654,E2 525.8054} C_DIS
LIN {X 27.4918,Y -130.0196,Z 165,A -77.3499,B 12.0249,C 0.2463,E1 12.0601,E2 527.7793} C_DIS
LIN {X 23.4369,Y -130.8108,Z 165,A -79.0304,B 12.0249,C 0.2449,E1 12.0555,E2 529.4486} C_DIS
LIN {X 19.9627,Y -131.3864,Z 165,A -80.625,B 12.0249,C 0.2478,E1 12.051,E2 531.0535} C_DIS
LIN {X 15.8832,Y -131.9413,Z 165,A -82.3086,B 12.0249,C 0.2464,E1 12.0464,E2 532.7271} C_DIS
LIN {X 12.5231,Y -132.3026,Z 165,A -83.8155,B 12.0249,C 0.2483,E1 12.0422,E2 534.2409} C_DIS
LIN {X 8.3124,Y -132.6338,Z 165,A -85.6164,B 12.0249,C 0.2484,E1 12.0372,E2 536.0404} C_DIS
LIN {X 4.4295,Y -132.822,Z 165,A -87.3781,B 12.0249,C 0.251,E1 12.0322,E2 537.8134} C_DIS
LIN {X 0.9669,Y -132.8884,Z 165,A -88.2416,B 12.0251,C 0.2353,E1 12.0301,E2 538.6008} C_DIS
Enddeposition()
LIN {X 0.9669,Y -132.8884,Z 165,A -88.2416,B 12.0251,C 0.2353,E1 12.0301,E2 538.6008} C_DIS
Startdeposition()
$VEL.CP = VEL_PRINT
LIN {X 3.4476,Y -133.7679,Z 165,A -86.8697,B 11.7259,C 0.2508,E1 11.7348,E2 537.3149} C_DIS
LIN {X 7.4151,Y -133.6083,Z 165,A -85.1128,B 11.7259,C 0.2489,E1 11.7397,E2 535.5501} C_DIS
LIN {X 11.5039,Y -133.3168,Z 165,A -83.4137,B 11.7259,C 0.2497,E1 11.7444,E2 533.8569} C_DIS
LIN {X 15.6993,Y -132.8879,Z 165,A -81.6455,B 11.7259,C 0.2498,E1 11.7493,E2 532.0923} C_DIS
LIN {X 19.6622,Y -132.3615,Z 165,A -79.8699,B 11.7259,C 0.2473,E1 11.7542,E2 530.3078} C_DIS
LIN {X 23.6313,Y -131.7087,Z 165,A -78.2236,B 11.7259,C 0.2481,E1 11.7587,E2 528.6697} C_DIS
LIN {X 27.7651,Y -130.9005,Z 165,A -76.4185,B 11.7259,C 0.2468,E1 11.7637,E2 526.8632} C_DIS
LIN {X 31.1356,Y -130.1392,Z 165,A -74.9659,B 11.7259,C 0.2463,E1 11.7676,E2 525.4129} C_DIS
LIN {X 37.917,Y -128.3276,Z 165,A -72.297,B 11.7259,C 0.2524,E1 11.7747,E2 522.7836} C_DIS
LIN {X 44.9586,Y -126.0337,Z 165,A -68.7539,B 11.7261,C 0.2393,E1 11.7842,E2 519.192} C_DIS
LIN {X 48.2636,Y -124.8048,Z 165,A -67.2556,B 11.7261,C 0.2379,E1 11.7881,E2 517.6939} C_DIS
LIN {X 52.0084,Y -123.2919,Z 165,A -65.4551,B 11.7262,C 0.2338,E1 11.7928,E2 515.8832} C_DIS
LIN {X 55.8704,Y -121.59,Z 165,A -63.8487,B 11.7262,C 0.2367,E1 11.7968,E2 514.3001} C_DIS
LIN {X 59.1064,Y -120.0499,Z 165,A -62.3529,B 11.7262,C 0.2356,E1 11.8006,E2 512.8077} C_DIS
LIN {X 61.8554,Y -118.6574,Z 165,A -60.943,B 11.7262,C 0.2313,E1 11.8041,E2 511.3854} C_DIS
LIN {X 65.6882,Y -116.5811,Z 165,A -59.0186,B 11.7264,C 0.2269,E1 11.8088,E2 509.4521} C_DIS
LIN {X 69.4893,Y -114.3564,Z 165,A -57.1431,B 11.7264,C 0.2241,E1 11.8133,E2 507.5761} C_DIS
LIN {X 72.5091,Y -112.4648,Z 165,A -55.2494,B 11.7266,C 0.2115,E1 11.8179,E2 505.635} C_DIS
LIN {X 76.0644,Y -110.0928,Z 165,A -53.7756,B 11.7266,C 0.2179,E1 11.8212,E2 504.2038} C_DIS
LIN {X 79.6574,Y -107.5214,Z 165,A -51.8327,B 11.7266,C 0.2131,E1 11.8256,E2 502.2527} C_DIS
LIN {X 83.2485,Y -104.7653,Z 165,A -49.4161,B 11.7269,C 0.1962,E1 11.831,E2 499.7743} C_DIS
LIN {X 87.3744,Y -101.3497,Z 165,A -47.7425,B 11.7267,C 0.2086,E1 11.8344,E2 498.1757} C_DIS
LIN {X 92.1853,Y -96.9952,Z 165,A -45.1397,B 11.7267,C 0.2076,E1 11.8397,E2 495.5918} C_DIS
LIN {X 96.8673,Y -92.3191,Z 165,A -42.1943,B 11.7269,C 0.1984,E1 11.8456,E2 492.6295} C_DIS
LIN {X 98.8979,Y -90.1407,Z 165,A -40.7322,B 11.7269,C 0.1904,E1 11.8484,E2 491.1427} C_DIS
LIN {X 103.1778,Y -85.2082,Z 165,A -38.1449,B 11.727,C 0.1896,E1 11.853,E2 488.5783} C_DIS
LIN {X 106.0329,Y -81.6288,Z 165,A -36.1689,B 11.727,C 0.1845,E1 11.8564,E2 486.5982} C_DIS
LIN {X 108.7062,Y -78.0325,Z 165,A -34.2904,B 11.7271,C 0.1809,E1 11.8595,E2 484.7224} C_DIS
LIN {X 111.2021,Y -74.4324,Z 165,A -32.4529,B 11.7271,C 0.1772,E1 11.8624,E2 482.8875} C_DIS
LIN {X 113.5966,Y -70.7239,Z 165,A -30.6217,B 11.7272,C 0.174,E1 11.8651,E2 481.0614} C_DIS
LIN {X 116.4701,Y -65.8857,Z 165,A -28.165,B 11.7274,C 0.1664,E1 11.8686,E2 478.5962} C_DIS
LIN {X 118.5447,Y -62.0701,Z 165,A -26.468,B 11.7274,C 0.166,E1 11.8708,E2 476.917} C_DIS
LIN {X 120.2214,Y -58.7586,Z 165,A -24.3731,B 11.7276,C 0.1476,E1 11.8734,E2 474.7575} C_DIS
LIN {X 122.0802,Y -54.7903,Z 165,A -23.0646,B 11.7275,C 0.1584,E1 11.8749,E2 473.5172} C_DIS
LIN {X 123.3727,Y -51.815,Z 165,A -21.6187,B 11.7275,C 0.1529,E1 11.8765,E2 472.0628} C_DIS
LIN {X 124.8321,Y -48.1934,Z 165,A -19.8872,B 11.7276,C 0.1466,E1 11.8782,E2 470.3219} C_DIS
LIN {X 126.2272,Y -44.4143,Z 165,A -17.8082,B 11.7278,C 0.1318,E1 11.8802,E2 468.197} C_DIS
LIN {X 127.5834,Y -40.3507,Z 165,A -16.3675,B 11.7278,C 0.1377,E1 11.8814,E2 466.803} C_DIS
LIN {X 129.9789,Y -31.8006,Z 165,A -12.6537,B 11.7278,C 0.1292,E1 11.8841,E2 463.0959} C_DIS
LIN {X 130.8308,Y -28.0877,Z 165,A -11.0824,B 11.7278,C 0.1262,E1 11.885,E2 461.5301} C_DIS
LIN {X 131.6622,Y -23.8911,Z 165,A -9.3284,B 11.7278,C 0.123,E1 11.886,E2 459.7836} C_DIS
LIN {X 132.2177,Y -20.5943,Z 165,A -7.9094,B 11.7279,C 0.1191,E1 11.8866,E2 458.3645} C_DIS
LIN {X 132.7345,Y -16.9524,Z 165,A -6.2245,B 11.7279,C 0.1114,E1 11.8872,E2 456.6644} C_DIS
LIN {X 133.1755,Y -13.0379,Z 165,A -4.6438,B 11.728,C 0.1094,E1 11.8877,E2 455.0949} C_DIS
LIN {X 133.5131,Y -8.971,Z 165,A -2.8297,B 11.728,C 0.1024,E1 11.8881,E2 453.2707} C_DIS
LIN {X 133.7145,Y -5.1103,Z 165,A -1.3034,B 11.728,C 0.1011,E1 11.8882,E2 451.7583} C_DIS
LIN {X 133.8093,Y -1.0017,Z 165,A 0.4017,B 11.7281,C 0.0975,E1 11.8883,E2 450.0581} C_DIS
LIN {X 133.7823,Y 2.9034,Z 165,A 2.162,B 11.7281,C 0.0901,E1 11.8883,E2 448.2852} C_DIS
LIN {X 133.6607,Y 6.3724,Z 165,A 3.5705,B 11.7281,C 0.0879,E1 11.8881,E2 446.8846} C_DIS
LIN {X 133.4217,Y 10.2248,Z 165,A 5.2743,B 11.7282,C 0.0816,E1 11.8877,E2 445.1729} C_DIS
LIN {X 133.0741,Y 14.0364,Z 165,A 6.8213,B 11.7282,C 0.0793,E1 11.8873,E2 443.6355} C_DIS
LIN {X 132.5974,Y 17.9983,Z 165,A 8.5088,B 11.7282,C 0.075,E1 11.8867,E2 441.9489} C_DIS
LIN {X 132.0059,Y 21.9109,Z 165,A 10.1326,B 11.7283,C 0.072,E1 11.886,E2 440.3321} C_DIS
LIN {X 131.4343,Y 25.1122,Z 165,A 11.5362,B 11.7283,C 0.0677,E1 11.8853,E2 438.9258} C_DIS
LIN {X 130.6191,Y 29.0656,Z 165,A 13.3786,B 11.7283,C 0.0595,E1 11.8842,E2 437.0678} C_DIS
LIN {X 129.5964,Y 33.3249,Z 165,A 15.4061,B 11.7284,C 0.05,E1 11.8828,E2 435.0199} C_DIS
LIN {X 128.6655,Y 36.7605,Z 165,A 17.0729,B 11.7284,C 0.0417,E1 11.8815,E2 433.3342} C_DIS
LIN {X 127.4545,Y 40.7544,Z 165,A 18.481,B 11.7284,C 0.0473,E1 11.8804,E2 431.971} C_DIS
LIN {X 126.0065,Y 45.034,Z 165,A 20.0785,B 11.7284,C 0.0513,E1 11.8789,E2 430.4131} C_DIS
LIN {X 125.1236,Y 47.4332,Z 165,A 21.4833,B 11.7284,C 0.0397,E1 11.8775,E2 428.9696} C_DIS
LIN {X 123.4807,Y 51.5563,Z 165,A 23.1062,B 11.7284,C 0.0422,E1 11.8759,E2 427.3789} C_DIS
LIN {X 122.2386,Y 54.4363,Z 165,A 24.5762,B 11.7284,C 0.0351,E1 11.8742,E2 425.8924} C_DIS
LIN {X 120.7723,Y 57.6159,Z 165,A 26.6563,B 11.7285,C 0.0151,E1 11.8716,E2 423.7399} C_DIS
LIN {X 118.5198,Y 62.1175,Z 165,A 28.0575,B 11.7285,C 0.0304,E1 11.8699,E2 422.4295} C_DIS
LIN {X 114.9933,Y 68.4296,Z 165,A 31.289,B 11.7285,C 0.0189,E1 11.8655,E2 419.1796} C_DIS
LIN {X 112.7858,Y 72.0101,Z 165,A 33.0905,B 11.7285,C 0.0144,E1 11.8628,E2 417.3769} C_DIS
LIN {X 110.7764,Y 75.0643,Z 165,A 34.5286,B 11.7285,C 0.0141,E1 11.8606,E2 415.9533} C_DIS
LIN {X 108.119,Y 78.8447,Z 165,A 36.6247,B 11.7285,C 0.0063,E1 11.8571,E2 413.8418} C_DIS
LIN {X 105.4547,Y 82.3741,Z 165,A 38.491,B 11.7285,C 0.0027,E1 11.854,E2 411.9777} C_DIS
LIN {X 102.7164,Y 85.7642,Z 165,A 40.3641,B 11.7285,C -0.0017,E1 11.8506,E2 410.1028} C_DIS
LIN {X 99.6877,Y 89.266,Z 165,A 42.2779,B 11.7285,C -0.0042,E1 11.8471,E2 408.1963} C_DIS
LIN {X 96.5849,Y 92.6146,Z 165,A 44.2369,B 11.7285,C -0.0084,E1 11.8434,E2 406.2359} C_DIS
LIN {X 93.4271,Y 95.7996,Z 165,A 46.1537,B 11.7285,C -0.0122,E1 11.8396,E2 404.3188} C_DIS
LIN {X 90.2223,Y 98.8239,Z 165,A 48.0358,B 11.7285,C -0.0157,E1 11.8357,E2 402.4366} C_DIS
LIN {X 86.9129,Y 101.7462,Z 165,A 49.9029,B 11.7285,C -0.0187,E1 11.8318,E2 400.5716} C_DIS
LIN {X 83.4779,Y 104.5827,Z 165,A 51.7846,B 11.7285,C -0.0214,E1 11.8277,E2 398.6924} C_DIS
LIN {X 79.8844,Y 107.3524,Z 165,A 53.6956,B 11.7285,C -0.024,E1 11.8234,E2 396.7847} C_DIS
LIN {X 76.1746,Y 110.0163,Z 165,A 55.5504,B 11.7285,C -0.0245,E1 11.8192,E2 394.9417} C_DIS
LIN {X 72.5881,Y 112.415,Z 165,A 57.4903,B 11.7285,C -0.0298,E1 11.8147,E2 392.9903} C_DIS
LIN {X 68.8184,Y 114.7616,Z 165,A 59.4521,B 11.7285,C -0.0342,E1 11.81,E2 391.0208} C_DIS
LIN {X 64.0121,Y 117.5097,Z 165,A 61.6997,B 11.7285,C -0.0343,E1 11.8045,E2 388.7879} C_DIS
LIN {X 60.0573,Y 119.5791,Z 165,A 63.6898,B 11.7285,C -0.0388,E1 11.7996,E2 386.7881} C_DIS
LIN {X 55.5824,Y 121.7232,Z 165,A 65.701,B 11.7285,C -0.0384,E1 11.7945,E2 384.7905} C_DIS
LIN {X 51.883,Y 123.3443,Z 165,A 67.4214,B 11.7285,C -0.0401,E1 11.7901,E2 383.0711} C_DIS
LIN {X 48.4835,Y 124.7193,Z 165,A 68.8848,B 11.7285,C -0.039,E1 11.7863,E2 381.6207} C_DIS
LIN {X 45.3998,Y 125.8746,Z 165,A 70.2857,B 11.7285,C -0.0402,E1 11.7827,E2 380.2209} C_DIS
LIN {X 42.3412,Y 126.9362,Z 165,A 71.6332,B 11.7285,C -0.0404,E1 11.7791,E2 378.8782} C_DIS
LIN {X 38.4289,Y 128.1771,Z 165,A 73.5808,B 11.7285,C -0.0466,E1 11.7739,E2 376.9081} C_DIS
LIN {X 34.6432,Y 129.2496,Z 165,A 75.1784,B 11.7285,C -0.0457,E1 11.7696,E2 375.3212} C_DIS
LIN {X 28.9241,Y 130.6503,Z 165,A 77.7866,B 11.7285,C -0.0494,E1 11.7625,E2 372.7031} C_DIS
LIN {X 25.031,Y 131.4499,Z 165,A 79.3614,B 11.7285,C -0.0471,E1 11.7582,E2 371.144} C_DIS
LIN {X 21.0482,Y 132.1474,Z 165,A 81.0678,B 11.7285,C -0.0472,E1 11.7535,E2 369.4411} C_DIS
LIN {X 17.4584,Y 132.6682,Z 165,A 82.5986,B 11.7285,C -0.0472,E1 11.7493,E2 367.9134} C_DIS
LIN {X 13.9741,Y 133.0808,Z 165,A 84.2034,B 11.7285,C -0.0502,E1 11.7448,E2 366.2968} C_DIS
LIN {X 9.9199,Y 133.4439,Z 165,A 85.831,B 11.7285,C -0.0477,E1 11.7403,E2 364.6837} C_DIS
LIN {X 6.5787,Y 133.6503,Z 165,A 87.338,B 11.7285,C -0.0496,E1 11.7361,E2 363.1684} C_DIS
LIN {X 2.3208,Y 133.792,Z 165,A 89.1626,B 11.7285,C -0.0496,E1 11.731,E2 361.3446} C_DIS
LIN {X -1.9465,Y 133.7982,Z 165,A 91.01,B 11.7285,C -0.05,E1 11.7258,E2 359.4957} C_DIS
LIN {X -6.0463,Y 133.6771,Z 165,A 92.8219,B 11.7285,C -0.0511,E1 11.7208,E2 357.678} C_DIS
LIN {X -9.8448,Y 133.4494,Z 165,A 94.3701,B 11.7285,C -0.0487,E1 11.7165,E2 356.1404} C_DIS
LIN {X -14.053,Y 133.0723,Z 165,A 96.1471,B 11.7285,C -0.0473,E1 11.7116,E2 354.3682} C_DIS
LIN {X -17.325,Y 132.6856,Z 165,A 97.6078,B 11.7285,C -0.0479,E1 11.7075,E2 352.9024} C_DIS
LIN {X -21.1327,Y 132.1343,Z 165,A 99.2948,B 11.7285,C -0.048,E1 11.7028,E2 351.2118} C_DIS
LIN {X -25.3626,Y 131.3865,Z 165,A 102.2629,B 11.7283,C -0.0739,E1 11.6944,E2 348.1085} C_DIS
LIN {X -33.1086,Y 129.6512,Z 165,A 104.4277,B 11.7284,C -0.0419,E1 11.6889,E2 346.0952} C_DIS
LIN {X -35.5537,Y 129.003,Z 165,A 106.5323,B 11.7284,C -0.0652,E1 11.6829,E2 343.8684} C_DIS
LIN {X -41.9852,Y 127.0547,Z 165,A 108.5659,B 11.7284,C -0.0425,E1 11.6778,E2 341.9389} C_DIS
LIN {X -46.3447,Y 125.5313,Z 165,A 110.5391,B 11.7284,C -0.0403,E1 11.6726,E2 339.9679} C_DIS
LIN {X -49.9539,Y 124.1376,Z 165,A 112.0908,B 11.7284,C -0.036,E1 11.6686,E2 338.4299} C_DIS
LIN {X -56.1455,Y 121.4628,Z 165,A 114.9775,B 11.7284,C -0.0324,E1 11.6612,E2 335.546} C_DIS
LIN {X -59.0223,Y 120.0913,Z 165,A 116.2782,B 11.7284,C -0.0291,E1 11.6579,E2 334.2541} C_DIS
LIN {X -65.994,Y 116.4087,Z 165,A 119.9127,B 11.7284,C -0.03,E1 11.649,E2 330.5921} C_DIS
LIN {X -69.9504,Y 114.0745,Z 165,A 121.854,B 11.7284,C -0.0264,E1 11.6443,E2 328.6557} C_DIS
LIN {X -73.7871,Y 111.6314,Z 165,A 123.7771,B 11.7284,C -0.0226,E1 11.6398,E2 326.7374} C_DIS
LIN {X -77.4046,Y 109.1545,Z 165,A 125.6942,B 11.7285,C -0.0202,E1 11.6354,E2 324.8175} C_DIS
LIN {X -80.8869,Y 106.5996,Z 165,A 127.5839,B 11.7285,C -0.0178,E1 11.6312,E2 322.9248} C_DIS
LIN {X -84.3715,Y 103.8637,Z 165,A 129.5256,B 11.7285,C -0.0152,E1 11.6269,E2 320.9796} C_DIS
LIN {X -87.7343,Y 101.0389,Z 165,A 131.4036,B 11.7285,C -0.0114,E1 11.623,E2 319.1039} C_DIS
LIN {X -91.012,Y 98.0966,Z 165,A 133.3039,B 11.7285,C -0.0079,E1 11.619,E2 317.2039} C_DIS
LIN {X -94.2167,Y 95.0226,Z 165,A 135.2147,B 11.7285,C -0.0041,E1 11.6152,E2 315.294} C_DIS
LIN {X -97.3982,Y 91.7587,Z 165,A 137.1509,B 11.7285,C 0.0005,E1 11.6115,E2 313.3618} C_DIS
LIN {X -100.3945,Y 88.4706,Z 165,A 139.0811,B 11.7285,C 0.0042,E1 11.6079,E2 311.4306} C_DIS
LIN {X -103.2492,Y 85.1219,Z 165,A 140.9885,B 11.7285,C 0.008,E1 11.6045,E2 309.5226} C_DIS
LIN {X -106.0153,Y 81.6516,Z 165,A 142.9621,B 11.7285,C 0.0109,E1 11.6011,E2 307.5423} C_DIS
LIN {X -108.6932,Y 78.0507,Z 165,A 144.8621,B 11.7285,C 0.016,E1 11.5979,E2 305.6471} C_DIS
LIN {X -111.1696,Y 74.481,Z 165,A 146.5952,B 11.7285,C 0.0234,E1 11.5952,E2 303.9313} C_DIS
LIN {X -114.3797,Y 69.4506,Z 165,A 149.1988,B 11.7285,C 0.0289,E1 11.5914,E2 301.3249} C_DIS
LIN {X -116.1133,Y 66.5119,Z 165,A 151.0539,B 11.7285,C 0.0241,E1 11.5887,E2 299.4242} C_DIS
LIN {X -117.7902,Y 63.4946,Z 165,A 152.388,B 11.7285,C 0.0311,E1 11.587,E2 298.1092} C_DIS
LIN {X -120.0244,Y 59.158,Z 165,A 154.2962,B 11.7285,C 0.0405,E1 11.5846,E2 296.2249} C_DIS
LIN {X -121.7452,Y 55.5348,Z 165,A 156.3971,B 11.7285,C 0.0369,E1 11.5821,E2 294.0801} C_DIS
LIN {X -123.1566,Y 52.3323,Z 165,A 157.7164,B 11.7285,C 0.0449,E1 11.5806,E2 292.7841} C_DIS
LIN {X -124.6428,Y 48.6802,Z 165,A 159.3045,B 11.7285,C 0.0517,E1 11.579,E2 291.21} C_DIS
LIN {X -125.7463,Y 45.7557,Z 165,A 160.6648,B 11.7284,C 0.055,E1 11.5777,E2 289.8485} C_DIS
LIN {X -126.8939,Y 42.4681,Z 165,A 162.1244,B 11.7284,C 0.0599,E1 11.5764,E2 288.3944} C_DIS
LIN {X -127.858,Y 39.4717,Z 165,A 163.4924,B 11.7284,C 0.0633,E1 11.5752,E2 287.0256} C_DIS
LIN {X -128.7597,Y 36.4237,Z 165,A 164.9443,B 11.7284,C 0.0652,E1 11.5741,E2 285.5644} C_DIS
LIN {X -129.888,Y 32.1758,Z 165,A 166.9032,B 11.7284,C 0.069,E1 11.5727,E2 283.5984} C_DIS
LIN {X -130.7464,Y 28.4785,Z 165,A 168.4712,B 11.7283,C 0.0749,E1 11.5718,E2 282.039} C_DIS
LIN {X -131.5678,Y 24.4143,Z 165,A 171.1287,B 11.7283,C 0.061,E1 11.5704,E2 279.2768} C_DIS
LIN {X -132.5657,Y 18.2331,Z 165,A 173.0366,B 11.7283,C 0.0856,E1 11.5697,E2 277.4658} C_DIS
LIN {X -133.022,Y 14.5202,Z 165,A 174.5988,B 11.7282,C 0.0912,E1 11.5692,E2 275.9101} C_DIS
LIN {X -133.3597,Y 10.9961,Z 165,A 176.1736,B 11.7282,C 0.0944,E1 11.5688,E2 274.3299} C_DIS
LIN {X -133.6268,Y 7.0471,Z 165,A 177.8602,B 11.7282,C 0.0995,E1 11.5685,E2 272.646} C_DIS
LIN {X -133.7686,Y 3.4224,Z 165,A 179.5307,B 11.7281,C 0.1016,E1 11.5683,E2 270.963} C_DIS
LIN {X -133.8116,Y -0.6599,Z 165,A -178.7517,B 11.7281,C 0.1074,E1 11.5683,E2 269.2511} C_DIS
LIN {X -133.7212,Y -4.9389,Z 165,A -176.9514,B 11.728,C 0.1135,E1 11.5685,E2 267.4566} C_DIS
LIN {X -133.5503,Y -8.3667,Z 165,A -175.4608,B 11.728,C 0.1174,E1 11.5687,E2 265.965} C_DIS
LIN {X -133.2319,Y -12.4511,Z 165,A -173.6538,B 11.728,C 0.1214,E1 11.5691,E2 264.1534} C_DIS
LIN {X -132.8363,Y -16.1322,Z 165,A -172.044,B 11.7279,C 0.1255,E1 11.5697,E2 262.5422} C_DIS
LIN {X -132.0586,Y -21.5946,Z 165,A -169.6887,B 11.7278,C 0.1325,E1 11.5706,E2 260.1901} C_DIS
LIN {X -130.6754,Y -28.8077,Z 165,A -166.5325,B 11.7277,C 0.1413,E1 11.5724,E2 257.0357} C_DIS
LIN {X -129.9663,Y -31.8529,Z 165,A -164.2801,B 11.7279,C 0.1252,E1 11.574,E2 254.6731} C_DIS
LIN {X -128.353,Y -37.8305,Z 165,A -162.4367,B 11.7276,C 0.1503,E1 11.5753,E2 252.9308} C_DIS
LIN {X -127.0751,Y -41.924,Z 165,A -160.5616,B 11.7276,C 0.1545,E1 11.5769,E2 251.0527} C_DIS
LIN {X -126.0161,Y -45.0074,Z 165,A -159.1728,B 11.7275,C 0.1585,E1 11.5782,E2 249.6659} C_DIS
LIN {X -124.8859,Y -48.0549,Z 165,A -157.7851,B 11.7275,C 0.1624,E1 11.5795,E2 248.2798} C_DIS
LIN {X -123.5832,Y -51.3109,Z 165,A -156.2489,B 11.7274,C 0.1657,E1 11.5812,E2 246.7407} C_DIS
LIN {X -121.8783,Y -55.2419,Z 165,A -154.2389,B 11.7274,C 0.1667,E1 11.5835,E2 244.7108} C_DIS
LIN {X -119.4296,Y -60.351,Z 165,A -151.9989,B 11.7272,C 0.1771,E1 11.5862,E2 242.4952} C_DIS
LIN {X -117.6766,Y -63.706,Z 165,A -150.182,B 11.7272,C 0.1769,E1 11.5886,E2 240.6557} C_DIS
LIN {X -115.4351,Y -67.6818,Z 165,A -148.2564,B 11.7272,C 0.1824,E1 11.5913,E2 238.7349} C_DIS
LIN {X -113.4231,Y -71.0028,Z 165,A -146.4972,B 11.7271,C 0.1844,E1 11.5939,E2 236.965} C_DIS
LIN {X -111.0266,Y -74.6947,Z 165,A -144.4867,B 11.7271,C 0.1861,E1 11.597,E2 234.9403} C_DIS
LIN {X -107.9772,Y -79.0382,Z 165,A -142.3465,B 11.7269,C 0.1943,E1 11.6005,E2 232.8177} C_DIS
LIN {X -105.2904,Y -82.5833,Z 165,A -140.4795,B 11.7269,C 0.1995,E1 11.6036,E2 230.9563} C_DIS
LIN {X -102.764,Y -85.7074,Z 165,A -138.6694,B 11.7269,C 0.2012,E1 11.6069,E2 229.1361} C_DIS
LIN {X -98.1093,Y -90.9982,Z 165,A -135.6323,B 11.7267,C 0.2072,E1 11.6125,E2 226.0981} C_DIS
LIN {X -94.9324,Y -94.3074,Z 165,A -133.6806,B 11.7267,C 0.2114,E1 11.6163,E2 224.1487} C_DIS
LIN {X -91.6891,Y -97.4639,Z 165,A -131.7393,B 11.7266,C 0.2151,E1 11.6202,E2 222.2078} C_DIS
LIN {X -88.4452,Y -100.4169,Z 165,A -129.8281,B 11.7266,C 0.2179,E1 11.6242,E2 220.2933} C_DIS
LIN {X -86.1176,Y -102.4199,Z 165,A -128.1718,B 11.7266,C 0.2124,E1 11.6279,E2 218.5954} C_DIS
LIN {X -83.052,Y -104.9216,Z 165,A -126.7773,B 11.7264,C 0.2223,E1 11.6308,E2 217.2383} C_DIS
LIN {X -80.3516,Y -107.0036,Z 165,A -125.3282,B 11.7264,C 0.225,E1 11.634,E2 215.791} C_DIS
LIN {X -77.4756,Y -109.1044,Z 165,A -123.6453,B 11.7264,C 0.2238,E1 11.6379,E2 214.089} C_DIS
LIN {X -73.2597,Y -111.9787,Z 165,A -121.5913,B 11.7263,C 0.2302,E1 11.6426,E2 212.0515} C_DIS
LIN {X -69.9067,Y -114.1013,Z 165,A -119.7126,B 11.7263,C 0.2284,E1 11.6472,E2 210.151} C_DIS
LIN {X -65.3769,Y -116.756,Z 165,A -117.7752,B 11.7261,C 0.2388,E1 11.6518,E2 208.2521} C_DIS
LIN {X -62.411,Y -118.3657,Z 165,A -116.2544,B 11.7261,C 0.2388,E1 11.6555,E2 206.7221} C_DIS
LIN {X -58.6004,Y -120.2995,Z 165,A -114.354,B 11.7261,C 0.2394,E1 11.6603,E2 204.8131} C_DIS
LIN {X -54.8888,Y -122.0362,Z 165,A -112.626,B 11.7261,C 0.242,E1 11.6647,E2 203.0883} C_DIS
LIN {X -51.7465,Y -123.4013,Z 165,A -111.1627,B 11.7261,C 0.2436,E1 11.6684,E2 201.6255} C_DIS
LIN {X -48.3364,Y -124.7765,Z 165,A -109.6406,B 11.726,C 0.2463,E1 11.6724,E2 200.1098} C_DIS
LIN {X -45.2262,Y -125.9372,Z 165,A -108.2504,B 11.726,C 0.2483,E1 11.676,E2 198.7233} C_DIS
LIN {X -41.4632,Y -127.2281,Z 165,A -106.3498,B 11.726,C 0.245,E1 11.6811,E2 196.7982} C_DIS
LIN {X -37.8361,Y -128.3513,Z 165,A -104.7933,B 11.726,C 0.2478,E1 11.6852,E2 195.2499} C_DIS
LIN {X -32.0791,Y -129.9118,Z 165,A -102.1285,B 11.726,C 0.2467,E1 11.6925,E2 192.5711} C_DIS
LIN {X -28.0756,Y -130.8334,Z 165,A -100.4658,B 11.7259,C 0.25,E1 11.697,E2 190.9199} C_DIS
LIN {X -23.8847,Y -131.6633,Z 165,A -98.6277,B 11.7259,C 0.2505,E1 11.702,E2 189.0802} C_DIS
LIN {X -19.9916,Y -132.311,Z 165,A -96.8762,B 11.7259,C 0.2496,E1 11.7069,E2 187.3205} C_DIS
LIN {X -16.1672,Y -132.8321,Z 165,A -95.2849,B 11.7259,C 0.2515,E1 11.7113,E2 185.7362} C_DIS
LIN {X -12.448,Y -133.2322,Z 165,A -93.6675,B 11.7259,C 0.2513,E1 11.7158,E2 184.1163} C_DIS
LIN {X -8.3899,Y -133.5489,Z 165,A -91.9623,B 11.7259,C 0.2524,E1 11.7205,E2 182.4151} C_DIS
LIN {X -4.4631,Y -133.7397,Z 165,A -90.1944,B 11.7259,C 0.2503,E1 11.7255,E2 180.636} C_DIS
LIN {X -0.6045,Y -133.8108,Z 165,A -88.6563,B 11.7259,C 0.253,E1 11.7297,E2 179.1113} C_DIS
LIN {X -0.6045,Y -133.8108,Z 165,A -88.6563,B 11.7259,C 0.253,E1 11.7297,E2 179.1113} C_DIS
Enddeposition()
LIN {X 0.9754,Y -134.7225,Z 165,A -88.2276,B 11.6439,C 0.2704,E1 11.6492,E2 178.7721} C_DIS
Startdeposition()
$VEL.CP = VEL_PRINT
LIN {X -2.16,Y -134.7129,Z 165,A -89.9303,B 11.6437,C 0.2798,E1 11.6443,E2 180.5213} C_DIS
LIN {X -6.4439,Y -134.5764,Z 165,A -91.7954,B 11.6437,C 0.2809,E1 11.639,E2 182.3924} C_DIS
LIN {X -10.1253,Y -134.3495,Z 165,A -93.3383,B 11.6437,C 0.2802,E1 11.6348,E2 183.9328} C_DIS
LIN {X -13.8716,Y -134.0152,Z 165,A -94.9459,B 11.6437,C 0.2802,E1 11.6303,E2 185.542} C_DIS
LIN {X -17.4813,Y -133.5911,Z 165,A -96.4307,B 11.6437,C 0.2783,E1 11.6262,E2 187.0198} C_DIS
LIN {X -20.6896,Y -133.132,Z 165,A -97.8664,B 11.6437,C 0.2793,E1 11.6222,E2 188.463} C_DIS
LIN {X -24.9374,Y -132.4025,Z 165,A -99.7057,B 11.6437,C 0.2787,E1 11.6171,E2 190.3037} C_DIS
LIN {X -28.4662,Y -131.6884,Z 165,A -101.2055,B 11.6437,C 0.2772,E1 11.6131,E2 191.8} C_DIS
LIN {X -32.3626,Y -130.7878,Z 165,A -103.1219,B 11.6437,C 0.2815,E1 11.6078,E2 193.7432} C_DIS
LIN {X -36.652,Y -129.6492,Z 165,A -104.7088,B 11.6438,C 0.273,E1 11.6036,E2 195.2935} C_DIS
LIN {X -39.2733,Y -128.8788,Z 165,A -106.0143,B 11.6438,C 0.2756,E1 11.6001,E2 196.6169} C_DIS
LIN {X -42.7819,Y -127.7571,Z 165,A -107.5215,B 11.6438,C 0.273,E1 11.5961,E2 198.117} C_DIS
LIN {X -46.0717,Y -126.6083,Z 165,A -108.981,B 11.6438,C 0.2712,E1 11.5922,E2 199.5739} C_DIS
LIN {X -49.1604,Y -125.4412,Z 165,A -110.4533,B 11.6438,C 0.2715,E1 11.5884,E2 201.0547} C_DIS
LIN {X -52.7712,Y -123.9672,Z 165,A -112.0523,B 11.644,C 0.2684,E1 11.5843,E2 202.6465} C_DIS
LIN {X -55.2591,Y -122.8763,Z 165,A -113.245,B 11.644,C 0.268,E1 11.5812,E2 203.8437} C_DIS
LIN {X -58.4551,Y -121.3889,Z 165,A -114.8516,B 11.644,C 0.2688,E1 11.5771,E2 205.4634} C_DIS
LIN {X -62.0951,Y -119.5686,Z 165,A -116.5756,B 11.644,C 0.2666,E1 11.5728,E2 207.1865} C_DIS
LIN {X -65.9349,Y -117.4956,Z 165,A -118.4478,B 11.644,C 0.2645,E1 11.5683,E2 209.0606} C_DIS
LIN {X -72.3718,Y -113.6444,Z 165,A -121.4073,B 11.6443,C 0.2547,E1 11.5613,E2 211.9915} C_DIS
LIN {X -74.8218,Y -112.046,Z 165,A -122.9273,B 11.6442,C 0.2591,E1 11.5576,E2 213.545} C_DIS
LIN {X -78.4947,Y -109.5044,Z 165,A -124.7882,B 11.6442,C 0.2552,E1 11.5534,E2 215.4009} C_DIS
LIN {X -81.8218,Y -107.0411,Z 165,A -126.6053,B 11.6442,C 0.2536,E1 11.5493,E2 217.2244} C_DIS
LIN {X -85.5704,Y -104.0696,Z 165,A -128.4839,B 11.6444,C 0.2465,E1 11.5453,E2 219.0834} C_DIS
LIN {X -87.905,Y -102.1044,Z 165,A -129.9705,B 11.6444,C 0.2484,E1 11.5421,E2 220.5926} C_DIS
LIN {X -91.3174,Y -99.0645,Z 165,A -131.9113,B 11.6444,C 0.2447,E1 11.5381,E2 222.5324} C_DIS
LIN {X -94.582,Y -95.953,Z 165,A -133.8662,B 11.6445,C 0.2418,E1 11.5341,E2 224.491} C_DIS
LIN {X -97.7218,Y -92.7536,Z 165,A -135.8258,B 11.6445,C 0.2391,E1 11.5303,E2 226.4562} C_DIS
LIN {X -100.8681,Y -89.3211,Z 165,A -137.7074,B 11.6447,C 0.2327,E1 11.5268,E2 228.3249} C_DIS
LIN {X -103.3934,Y -86.3858,Z 165,A -139.4092,B 11.6447,C 0.2303,E1 11.5237,E2 230.0326} C_DIS
LIN {X -105.9905,Y -83.1784,Z 165,A -141.1692,B 11.6448,C 0.2265,E1 11.5207,E2 231.7923} C_DIS
LIN {X -108.507,Y -79.8677,Z 165,A -143.0059,B 11.6448,C 0.224,E1 11.5176,E2 233.6363} C_DIS
LIN {X -111.0638,Y -76.2722,Z 165,A -144.7831,B 11.645,C 0.2174,E1 11.5148,E2 235.4003} C_DIS
LIN {X -113.0484,Y -73.2986,Z 165,A -146.4339,B 11.645,C 0.2166,E1 11.5122,E2 237.066} C_DIS
LIN {X -115.4967,Y -69.3779,Z 165,A -148.4511,B 11.645,C 0.2129,E1 11.5092,E2 239.0882} C_DIS
LIN {X -117.6813,Y -65.604,Z 165,A -150.3345,B 11.6452,C 0.2089,E1 11.5066,E2 240.9738} C_DIS
LIN {X -119.8305,Y -61.5874,Z 165,A -152.362,B 11.6452,C 0.2059,E1 11.504,E2 243.0107} C_DIS
LIN {X -121.9664,Y -57.2431,Z 165,A -154.2343,B 11.6454,C 0.1965,E1 11.5018,E2 244.8589} C_DIS
LIN {X -123.699,Y -53.3914,Z 165,A -156.0488,B 11.6454,C 0.1921,E1 11.4997,E2 246.6742} C_DIS
LIN {X -124.9791,Y -50.3221,Z 165,A -157.4772,B 11.6454,C 0.1886,E1 11.4982,E2 248.1032} C_DIS
LIN {X -126.2045,Y -47.165,Z 165,A -158.962,B 11.6455,C 0.1857,E1 11.4967,E2 249.5922} C_DIS
LIN {X -127.3605,Y -43.9483,Z 165,A -160.4159,B 11.6456,C 0.1817,E1 11.4954,E2 251.0449} C_DIS
LIN {X -128.4765,Y -40.5722,Z 165,A -161.9632,B 11.6456,C 0.1783,E1 11.494,E2 252.5951} C_DIS
LIN {X -129.4157,Y -37.4684,Z 165,A -163.9215,B 11.6456,C 0.1868,E1 11.4925,E2 254.6219} C_DIS
LIN {X -130.6299,Y -32.9846,Z 165,A -165.3674,B 11.6458,C 0.1699,E1 11.4915,E2 256.0024} C_DIS
LIN {X -131.4262,Y -29.6551,Z 165,A -166.8958,B 11.6458,C 0.1673,E1 11.4905,E2 257.5382} C_DIS
LIN {X -132.625,Y -23.7231,Z 165,A -169.1,B 11.646,C 0.1521,E1 11.4894,E2 259.6953} C_DIS
LIN {X -133.0795,Y -21.0283,Z 165,A -170.6726,B 11.646,C 0.1575,E1 11.4886,E2 261.3164} C_DIS
LIN {X -133.5209,Y -18.0171,Z 165,A -171.9911,B 11.646,C 0.1542,E1 11.4881,E2 262.6367} C_DIS
LIN {X -133.9862,Y -14.1413,Z 165,A -173.6749,B 11.646,C 0.1499,E1 11.4876,E2 264.3216} C_DIS
LIN {X -134.3617,Y -9.9585,Z 165,A -175.4191,B 11.6461,C 0.1438,E1 11.4872,E2 266.059} C_DIS
LIN {X -134.5728,Y -6.5156,Z 165,A -176.927,B 11.6461,C 0.1403,E1 11.4869,E2 267.5702} C_DIS
LIN {X -134.7088,Y -2.4086,Z 165,A -178.6819,B 11.6462,C 0.1353,E1 11.4869,E2 269.3242} C_DIS
LIN {X -134.7242,Y 1.4722,Z 165,A 179.5192,B 11.6462,C 0.1336,E1 11.4869,E2 271.1393} C_DIS
LIN {X -134.62,Y 5.4514,Z 165,A 177.9046,B 11.6463,C 0.127,E1 11.4869,E2 272.7426} C_DIS
LIN {X -134.3739,Y 9.7904,Z 165,A 175.9812,B 11.6463,C 0.1231,E1 11.4873,E2 274.673} C_DIS
LIN {X -133.9661,Y 14.3281,Z 165,A 174.0759,B 11.6464,C 0.1167,E1 11.4878,E2 276.5723} C_DIS
LIN {X -133.5403,Y 17.8688,Z 165,A 172.5009,B 11.6464,C 0.1135,E1 11.4884,E2 278.1527} C_DIS
LIN {X -132.7606,Y 22.9622,Z 165,A 170.4127,B 11.6465,C 0.105,E1 11.4893,E2 280.2261} C_DIS
LIN {X -131.942,Y 27.2695,Z 165,A 168.4959,B 11.6465,C 0.1006,E1 11.4903,E2 282.1469} C_DIS
LIN {X -131.22,Y 30.5578,Z 165,A 166.9657,B 11.6465,C 0.0986,E1 11.4913,E2 283.6873} C_DIS
LIN {X -130.3522,Y 34.0716,Z 165,A 165.3083,B 11.6466,C 0.0966,E1 11.4924,E2 285.3572} C_DIS
LIN {X -129.3233,Y 37.7837,Z 165,A 163.7885,B 11.6466,C 0.0895,E1 11.4936,E2 286.8609} C_DIS
LIN {X -128.3507,Y 40.9659,Z 165,A 162.3756,B 11.6466,C 0.0854,E1 11.4948,E2 288.2719} C_DIS
LIN {X -127.316,Y 44.0766,Z 165,A 160.9336,B 11.6467,C 0.0825,E1 11.4961,E2 289.718} C_DIS
LIN {X -126.1559,Y 47.2949,Z 165,A 159.4506,B 11.6467,C 0.079,E1 11.4975,E2 291.2026} C_DIS
LIN {X -124.8533,Y 50.6342,Z 165,A 157.919,B 11.6467,C 0.075,E1 11.4991,E2 292.7334} C_DIS
LIN {X -123.6169,Y 53.5813,Z 165,A 156.5291,B 11.6467,C 0.0719,E1 11.5006,E2 294.1253} C_DIS
LIN {X -122.1778,Y 56.7867,Z 165,A 154.9537,B 11.6468,C 0.0696,E1 11.5024,E2 295.7088} C_DIS
LIN {X -120.6228,Y 60.0202,Z 165,A 153.4872,B 11.6468,C 0.0642,E1 11.5042,E2 297.1664} C_DIS
LIN {X -119.1603,Y 62.8727,Z 165,A 152.1367,B 11.6468,C 0.0603,E1 11.506,E2 298.5138} C_DIS
LIN {X -116.1118,Y 68.3423,Z 165,A 149.0154,B 11.6468,C 0.0632,E1 11.5104,E2 301.6865} C_DIS
LIN {X -114.1174,Y 71.6229,Z 165,A 147.6794,B 11.6468,C 0.0527,E1 11.5123,E2 302.9855} C_DIS
LIN {X -112.0102,Y 74.8755,Z 165,A 146.0154,B 11.6469,C 0.0489,E1 11.5148,E2 304.6495} C_DIS
LIN {X -109.6896,Y 78.2357,Z 165,A 144.305,B 11.6469,C 0.0441,E1 11.5176,E2 306.3549} C_DIS
LIN {X -107.2334,Y 81.5704,Z 165,A 142.4428,B 11.6469,C 0.0421,E1 11.5207,E2 308.2271} C_DIS
LIN {X -104.3466,Y 85.2314,Z 165,A 140.4782,B 11.6469,C 0.037,E1 11.5241,E2 310.1873} C_DIS
LIN {X -101.6232,Y 88.4611,Z 165,A 138.65,B 11.6469,C 0.0336,E1 11.5274,E2 312.0172} C_DIS
LIN {X -98.5396,Y 91.8834,Z 165,A 136.6847,B 11.6469,C 0.0294,E1 11.5312,E2 313.9812} C_DIS
LIN {X -95.3833,Y 95.1562,Z 165,A 134.7426,B 11.6469,C 0.0254,E1 11.5349,E2 315.9221} C_DIS
LIN {X -92.2539,Y 98.1932,Z 165,A 132.8498,B 11.6469,C 0.0224,E1 11.5388,E2 317.8175} C_DIS
LIN {X -88.9019,Y 101.2385,Z 165,A 130.8862,B 11.6469,C 0.0194,E1 11.5429,E2 319.7836} C_DIS
LIN {X -85.5713,Y 104.0688,Z 165,A 129.0419,B 11.6469,C 0.0154,E1 11.5468,E2 321.6243} C_DIS
LIN {X -82.1305,Y 106.805,Z 165,A 127.1188,B 11.6469,C 0.0131,E1 11.551,E2 323.5519} C_DIS
LIN {X -78.5117,Y 109.4922,Z 165,A 125.2061,B 11.647,C 0.0096,E1 11.5554,E2 325.4621} C_DIS
LIN {X -74.7099,Y 112.1208,Z 165,A 123.2594,B 11.647,C 0.0058,E1 11.5598,E2 327.4047} C_DIS
LIN {X -70.8785,Y 114.5818,Z 165,A 121.2819,B 11.647,C 0.0036,E1 11.5645,E2 329.3852} C_DIS
LIN {X -67.2147,Y 116.7686,Z 165,A 119.4495,B 11.647,C 0.0012,E1 11.5689,E2 331.218} C_DIS
LIN {X -62.3842,Y 119.4167,Z 165,A 117.2558,B 11.647,C -0.0056,E1 11.5743,E2 333.3918} C_DIS
LIN {X -59.5334,Y 120.863,Z 165,A 115.8497,B 11.647,C -0.0064,E1 11.5778,E2 334.8022} C_DIS
LIN {X -56.3058,Y 122.4002,Z 165,A 114.1961,B 11.647,C -0.0053,E1 11.582,E2 336.4703} C_DIS
LIN {X -51.5579,Y 124.475,Z 165,A 112.1459,B 11.647,C -0.0115,E1 11.5872,E2 338.5005} C_DIS
LIN {X -48.7925,Y 125.5842,Z 165,A 110.8072,B 11.647,C -0.0113,E1 11.5907,E2 339.8466} C_DIS
LIN {X -45.5576,Y 126.7937,Z 165,A 109.3321,B 11.647,C -0.0127,E1 11.5946,E2 341.3213} C_DIS
LIN {X -41.9361,Y 128.0387,Z 165,A 107.4983,B 11.647,C -0.0096,E1 11.5995,E2 343.1783} C_DIS
LIN {X -35.109,Y 130.0756,Z 165,A 104.8295,B 11.647,C -0.0206,E1 11.6066,E2 345.802} C_DIS
LIN {X -31.1694,Y 131.0755,Z 165,A 102.8926,B 11.647,C -0.0171,E1 11.6119,E2 347.7625} C_DIS
LIN {X -25.5631,Y 132.2829,Z 165,A 100.7016,B 11.647,C -0.0245,E1 11.6178,E2 349.9223} C_DIS
LIN {X -22.7086,Y 132.8036,Z 165,A 99.1509,B 11.647,C -0.0178,E1 11.6221,E2 351.5099} C_DIS
LIN {X -19.0384,Y 133.3781,Z 165,A 97.6669,B 11.647,C -0.0208,E1 11.6262,E2 352.9815} C_DIS
LIN {X -15.2027,Y 133.8718,Z 165,A 95.8811,B 11.647,C -0.0181,E1 11.6312,E2 354.7833} C_DIS
LIN {X -11.3246,Y 134.2533,Z 165,A 94.3562,B 11.647,C -0.0218,E1 11.6354,E2 356.2915} C_DIS
LIN {X -7.8304,Y 134.5032,Z 165,A 92.7974,B 11.647,C -0.0205,E1 11.6397,E2 357.8577} C_DIS
LIN {X -3.5612,Y 134.6833,Z 165,A 90.9963,B 11.647,C -0.0212,E1 11.6448,E2 359.656} C_DIS
LIN {X 0.6607,Y 134.7287,Z 165,A 89.2341,B 11.647,C -0.0221,E1 11.6497,E2 361.4133} C_DIS
LIN {X 4.3598,Y 134.6611,Z 165,A 87.7061,B 11.647,C -0.0232,E1 11.6539,E2 362.9353} C_DIS
LIN {X 8.026,Y 134.4911,Z 165,A 86.1003,B 11.647,C -0.022,E1 11.6584,E2 364.5458} C_DIS
LIN {X 11.6961,Y 134.222,Z 165,A 84.4236,B 11.647,C -0.019,E1 11.6631,E2 366.2352} C_DIS
LIN {X 15.8997,Y 133.7886,Z 165,A 82.7651,B 11.647,C -0.0219,E1 11.6677,E2 367.8765} C_DIS
LIN {X 19.8233,Y 133.2659,Z 165,A 80.9405,B 11.647,C -0.0178,E1 11.6728,E2 369.7176} C_DIS
LIN {X 23.8801,Y 132.5969,Z 165,A 79.3433,B 11.647,C -0.0207,E1 11.6771,E2 371.2962} C_DIS
LIN {X 27.1339,Y 131.9696,Z 165,A 77.8909,B 11.647,C -0.0189,E1 11.6811,E2 372.7533} C_DIS
LIN {X 31.6659,Y 130.9558,Z 165,A 75.935,B 11.647,C -0.0182,E1 11.6864,E2 374.7066} C_DIS
LIN {X 34.8673,Y 130.14,Z 165,A 74.5119,B 11.647,C -0.0168,E1 11.6903,E2 376.1316} C_DIS
LIN {X 38.3611,Y 129.1543,Z 165,A 72.9548,B 11.647,C -0.0153,E1 11.6944,E2 377.6901} C_DIS
LIN {X 41.5819,Y 128.154,Z 165,A 71.593,B 11.647,C -0.0159,E1 11.698,E2 379.043} C_DIS
LIN {X 45.5475,Y 126.7973,Z 165,A 69.8129,B 11.647,C -0.0143,E1 11.7027,E2 380.8227} C_DIS
LIN {X 49.0331,Y 125.4907,Z 165,A 68.2453,B 11.647,C -0.0131,E1 11.7068,E2 382.3883} C_DIS
LIN {X 52.1804,Y 124.215,Z 165,A 66.7992,B 11.647,C -0.0115,E1 11.7106,E2 383.8347} C_DIS
LIN {X 55.3272,Y 122.8459,Z 165,A 65.3545,B 11.647,C -0.0103,E1 11.7142,E2 385.2776} C_DIS
LIN {X 58.3443,Y 121.4418,Z 165,A 63.987,B 11.647,C -0.0098,E1 11.7177,E2 386.6394} C_DIS
LIN {X 61.1804,Y 120.0376,Z 165,A 62.409,B 11.647,C -0.0021,E1 11.7217,E2 388.2453} C_DIS
LIN {X 64.4611,Y 118.3106,Z 165,A 60.2208,B 11.647,C 0.0156,E1 11.7273,E2 390.5064} C_DIS
LIN {X 69.6532,Y 115.3302,Z 165,A 58.792,B 11.647,C -0.0094,E1 11.7304,E2 391.8023} C_DIS
LIN {X 73.5927,Y 112.8574,Z 165,A 56.4135,B 11.647,C 0.0041,E1 11.7361,E2 394.2293} C_DIS
LIN {X 77.3812,Y 110.2945,Z 165,A 54.4993,B 11.647,C 0.0064,E1 11.7405,E2 396.1402} C_DIS
LIN {X 80.8487,Y 107.7787,Z 165,A 52.6705,B 11.647,C 0.0097,E1 11.7446,E2 397.9703} C_DIS
LIN {X 84.4475,Y 104.9822,Z 165,A 50.7684,B 11.647,C 0.0122,E1 11.7487,E2 399.8686} C_DIS
LIN {X 87.9461,Y 102.0691,Z 165,A 48.8566,B 11.647,C 0.0151,E1 11.7528,E2 401.7781} C_DIS
LIN {X 91.3078,Y 99.0734,Z 165,A 47.0084,B 11.647,C 0.0171,E1 11.7566,E2 403.619} C_DIS
LIN {X 94.4546,Y 96.0779,Z 165,A 45.1329,B 11.647,C 0.0215,E1 11.7604,E2 405.4986} C_DIS
LIN {X 97.6542,Y 92.8246,Z 165,A 43.1869,B 11.647,C 0.0257,E1 11.7642,E2 407.4462} C_DIS
LIN {X 100.7075,Y 89.5027,Z 165,A 41.2757,B 11.647,C 0.0296,E1 11.7678,E2 409.3574} C_DIS
LIN {X 103.6616,Y 86.0634,Z 165,A 39.4103,B 11.647,C 0.0322,E1 11.7711,E2 411.2162} C_DIS
LIN {X 106.3353,Y 82.7374,Z 165,A 37.5813,B 11.647,C 0.0367,E1 11.7743,E2 413.0479} C_DIS
LIN {X 109.0635,Y 79.1061,Z 165,A 35.2441,B 11.6469,C 0.052,E1 11.7782,E2 415.435} C_DIS
LIN {X 111.6773,Y 75.3712,Z 165,A 33.8581,B 11.6469,C 0.0418,E1 11.7803,E2 416.7557} C_DIS
LIN {X 113.7929,Y 72.1378,Z 165,A 32.1201,B 11.6469,C 0.0484,E1 11.7829,E2 418.5061} C_DIS
LIN {X 116.1574,Y 68.2647,Z 165,A 30.0663,B 11.6469,C 0.0566,E1 11.7859,E2 420.5762} C_DIS
LIN {X 118.5123,Y 64.0904,Z 165,A 28.206,B 11.6469,C 0.057,E1 11.7884,E2 422.4165} C_DIS
LIN {X 120.4361,Y 60.3976,Z 165,A 26.2807,B 11.6469,C 0.0657,E1 11.7909,E2 424.3617} C_DIS
LIN {X 122.3651,Y 56.3818,Z 165,A 24.6731,B 11.6469,C 0.0629,E1 11.7927,E2 425.936} C_DIS
LIN {X 123.8602,Y 53.0188,Z 165,A 23.1758,B 11.6469,C 0.0652,E1 11.7944,E2 427.4263} C_DIS
LIN {X 125.0579,Y 50.1267,Z 165,A 21.7597,B 11.6468,C 0.0712,E1 11.7959,E2 428.8538} C_DIS
LIN {X 127.1453,Y 44.5691,Z 165,A 19.4753,B 11.6468,C 0.0715,E1 11.7981,E2 431.1111} C_DIS
LIN {X 129.8314,Y 36.0004,Z 165,A 15.5157,B 11.6467,C 0.0861,E1 11.8014,E2 435.0914} C_DIS
LIN {X 130.9254,Y 31.7919,Z 165,A 13.7172,B 11.6467,C 0.0899,E1 11.8026,E2 436.8855} C_DIS
LIN {X 131.6917,Y 28.451,Z 165,A 12.289,B 11.6467,C 0.0933,E1 11.8034,E2 438.3114} C_DIS
LIN {X 132.3869,Y 25.0192,Z 165,A 10.8003,B 11.6467,C 0.0976,E1 11.8042,E2 439.8014} C_DIS
LIN {X 133.1288,Y 20.71,Z 165,A 8.9492,B 11.6466,C 0.1027,E1 11.8051,E2 441.6533} C_DIS
LIN {X 133.6324,Y 17.1663,Z 165,A 7.4292,B 11.6466,C 0.1071,E1 11.8057,E2 443.1746} C_DIS
LIN {X 134.0989,Y 13.0273,Z 165,A 5.7348,B 11.6465,C 0.1102,E1 11.8062,E2 444.8614} C_DIS
LIN {X 134.3952,Y 9.499,Z 165,A 4.1376,B 11.6465,C 0.1171,E1 11.8065,E2 446.4714} C_DIS
LIN {X 134.6281,Y 5.2449,Z 165,A 2.4833,B 11.6465,C 0.1181,E1 11.8067,E2 448.1083} C_DIS
LIN {X 134.7182,Y 1.8442,Z 165,A 1.0323,B 11.6464,C 0.1225,E1 11.8068,E2 449.5613} C_DIS
LIN {X 134.7117,Y -2.2324,Z 165,A -0.6971,B 11.6464,C 0.1275,E1 11.8068,E2 451.292} C_DIS
LIN {X 134.5764,Y -6.4439,Z 165,A -2.5244,B 11.6462,C 0.1337,E1 11.8066,E2 453.1256} C_DIS
LIN {X 134.3495,Y -10.1253,Z 165,A -3.9585,B 11.6462,C 0.1346,E1 11.8063,E2 454.5449} C_DIS
LIN {X 134.0561,Y -13.4727,Z 165,A -5.5323,B 11.6462,C 0.1429,E1 11.8059,E2 456.1381} C_DIS
LIN {X 133.5822,Y -17.5497,Z 165,A -7.1235,B 11.6462,C 0.1437,E1 11.8053,E2 457.7123} C_DIS
LIN {X 133.1055,Y -20.8606,Z 165,A -8.5618,B 11.6461,C 0.1483,E1 11.8047,E2 459.1541} C_DIS
LIN {X 132.5488,Y -24.1485,Z 165,A -9.8838,B 11.6461,C 0.1498,E1 11.8041,E2 460.466} C_DIS
LIN {X 131.9837,Y -27.0648,Z 165,A -11.2273,B 11.646,C 0.1557,E1 11.8034,E2 461.8207} C_DIS
LIN {X 131.0074,Y -31.4518,Z 165,A -13.1432,B 11.646,C 0.1614,E1 11.8022,E2 463.7394} C_DIS
LIN {X 129.6811,Y -36.5379,Z 165,A -15.2992,B 11.6458,C 0.1656,E1 11.8006,E2 465.8882} C_DIS
LIN {X 128.4676,Y -40.6001,Z 165,A -17.078,B 11.6458,C 0.1701,E1 11.7992,E2 467.6662} C_DIS
LIN {X 127.3427,Y -43.9996,Z 165,A -18.4689,B 11.6458,C 0.1707,E1 11.7979,E2 469.0426} C_DIS
LIN {X 126.4562,Y -46.4897,Z 165,A -20.1236,B 11.6455,C 0.1886,E1 11.7963,E2 470.7638} C_DIS
LIN {X 125.0124,Y -50.2395,Z 165,A -21.0972,B 11.6457,C 0.173,E1 11.7954,E2 471.649} C_DIS
LIN {X 123.1698,Y -54.603,Z 165,A -23.5077,B 11.6455,C 0.1896,E1 11.7927,E2 474.1107} C_DIS
LIN {X 121.3593,Y -58.5169,Z 165,A -25.1641,B 11.6455,C 0.1896,E1 11.7907,E2 475.7474} C_DIS
LIN {X 119.6467,Y -61.9463,Z 165,A -26.806,B 11.6455,C 0.1943,E1 11.7886,E2 477.3927} C_DIS
LIN {X 117.6654,Y -65.6326,Z 165,A -28.6715,B 11.6453,C 0.2014,E1 11.7861,E2 479.2709} C_DIS
LIN {X 115.4097,Y -69.5216,Z 165,A -30.364,B 11.6453,C 0.2004,E1 11.7838,E2 480.9386} C_DIS
LIN {X 113.4744,Y -72.6374,Z 165,A -32.0618,B 11.6452,C 0.2081,E1 11.7812,E2 482.6552} C_DIS
LIN {X 111.1976,Y -76.0773,Z 165,A -33.8099,B 11.6451,C 0.2124,E1 11.7785,E2 484.4045} C_DIS
LIN {X 108.6228,Y -79.7101,Z 165,A -35.6388,B 11.6451,C 0.2153,E1 11.7755,E2 486.2277} C_DIS
LIN {X 106.0724,Y -83.074,Z 165,A -37.4613,B 11.645,C 0.2204,E1 11.7724,E2 488.0555} C_DIS
LIN {X 103.2739,Y -86.5282,Z 165,A -40.3282,B 11.6443,C 0.2512,E1 11.7671,E2 491.0438} C_DIS
LIN {X 98.2277,Y -92.2173,Z 165,A -42.5341,B 11.6448,C 0.2308,E1 11.7631,E2 493.1278} C_DIS
LIN {X 93.3087,Y -97.1915,Z 165,A -45.3232,B 11.6448,C 0.2322,E1 11.7576,E2 495.8972} C_DIS
LIN {X 88.4478,Y -101.6348,Z 165,A -48.2325,B 11.6445,C 0.241,E1 11.7515,E2 498.8231} C_DIS
LIN {X 85.1396,Y -104.4217,Z 165,A -50.1236,B 11.6445,C 0.246,E1 11.7475,E2 500.7224} C_DIS
LIN {X 79.016,Y -109.1287,Z 165,A -53.1755,B 11.6445,C 0.246,E1 11.7407,E2 503.749} C_DIS
LIN {X 75.9562,Y -111.2806,Z 165,A -55.1988,B 11.6441,C 0.2603,E1 11.7359,E2 505.8273} C_DIS
LIN {X 72.818,Y -113.3587,Z 165,A -56.7085,B 11.6441,C 0.2606,E1 11.7324,E2 507.3273} C_DIS
LIN {X 69.9578,Y -115.146,Z 165,A -57.6061,B 11.6444,C 0.2487,E1 11.7304,E2 508.16} C_DIS
LIN {X 67.5169,Y -116.5937,Z 165,A -59.1166,B 11.6442,C 0.2588,E1 11.7267,E2 509.7093} C_DIS
LIN {X 63.6198,Y -118.7652,Z 165,A -61.0756,B 11.6441,C 0.2633,E1 11.7219,E2 511.6777} C_DIS
LIN {X 59.8328,Y -120.7153,Z 165,A -62.7707,B 11.6441,C 0.2628,E1 11.7177,E2 513.3599} C_DIS
LIN {X 56.5335,Y -122.2949,Z 165,A -64.2158,B 11.6441,C 0.2621,E1 11.7141,E2 514.7928} C_DIS
LIN {X 53.2841,Y -123.7454,Z 165,A -65.7334,B 11.6441,C 0.2642,E1 11.7102,E2 516.3122} C_DIS
LIN {X 50.0777,Y -125.0777,Z 165,A -67.1783,B 11.6441,C 0.2652,E1 11.7065,E2 517.7545} C_DIS
LIN {X 47.2443,Y -126.1748,Z 165,A -68.4007,B 11.6441,C 0.2649,E1 11.7033,E2 518.9693} C_DIS
LIN {X 43.552,Y -127.4978,Z 165,A -70.8545,B 11.6435,C 0.287,E1 11.6966,E2 521.5212} C_DIS
LIN {X 38.454,Y -129.1271,Z 165,A -72.3474,B 11.6439,C 0.2691,E1 11.6928,E2 522.9196} C_DIS
LIN {X 33.4707,Y -130.5066,Z 165,A -74.6113,B 11.6439,C 0.2728,E1 11.6867,E2 525.1932} C_DIS
LIN {X 29.8637,Y -131.3786,Z 165,A -76.2368,B 11.6438,C 0.2752,E1 11.6822,E2 526.8256} C_DIS
LIN {X 26.205,Y -132.1586,Z 165,A -77.9013,B 11.6438,C 0.2783,E1 11.6777,E2 528.5003} C_DIS
LIN {X 22.2549,Y -132.8793,Z 165,A -79.4803,B 11.6438,C 0.2761,E1 11.6734,E2 530.0646} C_DIS
Enddeposition()
END
